LIN {X 0,Y 474.587,Z 604.783,A -85,B 0,C 180,E1 6633.911,E2 6633.911} C_VEL
LIN {X 0,Y 484.461,Z 641.921,A -85,B 0,C 180,E1 6635.452,E2 6635.452} C_VEL
LIN {X 0,Y 481.473,Z 693.679,A -85,B 0,C 180,E1 6638.347,E2 6638.347} C_VEL
LIN {X 0,Y 478.667,Z 736.366,A -85,B 0,C 180,E1 6642.712,E2 6642.712} C_VEL
LIN {X 0,Y 476.602,Z 767.326,A -85,B 0,C 180,E1 6648.057,E2 6648.057} C_VEL
LIN {X 0,Y 475.424,Z 786.828,A -85,B 0,C 180,E1 6654.507,E2 6654.507} C_VEL
LIN {X 0,Y 475.028,Z 791.676,A -85,B 0,C 180,E1 6660.917,E2 6660.917} C_VEL
LIN {X 0,Y 475.519,Z 782.888,A -85,B 0,C 180,E1 6667.335,E2 6667.335} C_VEL
LIN {X 0,Y 477.046,Z 759.466,A -85,B 0,C 180,E1 6673.569,E2 6673.569} C_VEL
LIN {X 0,Y 479.555,Z 723.123,A -85,B 0,C 180,E1 6678.814,E2 6678.814} C_VEL
LIN {X 0,Y 482.628,Z 675.847,A -85,B 0,C 180,E1 6682.718,E2 6682.718} C_VEL
LIN {X 0,Y 482.433,Z 629.842,A -85,B 0,C 180,E1 6684.849,E2 6684.849} C_VEL
LIN {X 0,Y 474.42,Z 602.81,A -85,B 0,C 180,E1 6686.158,E2 6686.158} C_VEL
LIN {X 0,Y 474.205,Z 602.81,A -85,B 0,C 180,E1 6696.301,E2 6696.301} C_VEL
LIN {X 0,Y 474.043,Z 602.81,A -85,B 0,C 180,E1 6706.534,E2 6706.534} C_VEL
LIN {X 0,Y 473.963,Z 602.81,A -85,B 0,C 180,E1 6707.161,E2 6707.161} C_VEL
LIN {X 0,Y 465.924,Z 602.81,A -85,B 0,C 180,E1 6711.395,E2 6711.395} C_VEL
LIN {X 0,Y 466.396,Z 602.81,A -85,B 0,C 180,E1 6721.87,E2 6721.87} C_VEL
LIN {X 0,Y 466.767,Z 604.8,A -85,B 0,C 180,E1 6722.959,E2 6722.959} C_VEL
LIN {X 0,Y 476.808,Z 643.163,A -85,B 0,C 180,E1 6724.21,E2 6724.21} C_VEL
LIN {X 0,Y 475.259,Z 703.396,A -85,B 0,C 180,E1 6725.752,E2 6725.752} C_VEL
LIN {X 0,Y 472.339,Z 755.137,A -85,B 0,C 180,E1 6729.032,E2 6729.032} C_VEL
LIN {X 0,Y 469.648,Z 797.381,A -85,B 0,C 180,E1 6733.842,E2 6733.842} C_VEL
LIN {X 0,Y 468.095,Z 827.68,A -85,B 0,C 180,E1 6739.745,E2 6739.745} C_VEL
LIN {X 0,Y 467.651,Z 842.415,A -85,B 0,C 180,E1 6745.362,E2 6745.362} C_VEL
LIN {X 0,Y 467.519,Z 845.96,A -85,B 0,C 180,E1 6750.945,E2 6750.945} C_VEL
LIN {X 0,Y 467.394,Z 838.979,A -85,B 0,C 180,E1 6756.54,E2 6756.54} C_VEL
LIN {X 0,Y 468.068,Z 818.515,A -85,B 0,C 180,E1 6762.593,E2 6762.593} C_VEL
LIN {X 0,Y 470.107,Z 786.148,A -85,B 0,C 180,E1 6767.872,E2 6767.872} C_VEL
LIN {X 0,Y 473.479,Z 740.316,A -85,B 0,C 180,E1 6772.26,E2 6772.26} C_VEL
LIN {X 0,Y 476.388,Z 687.666,A -85,B 0,C 180,E1 6774.942,E2 6774.942} C_VEL
LIN {X 0,Y 475.283,Z 629.797,A -85,B 0,C 180,E1 6776.245,E2 6776.245} C_VEL
LIN {X 0,Y 466.568,Z 602.81,A -85,B 0,C 180,E1 6777.358,E2 6777.358} C_VEL
LIN {X 0,Y 466.192,Z 602.81,A -85,B 0,C 180,E1 6787.107,E2 6787.107} C_VEL
LIN {X 0,Y 466.037,Z 602.81,A -85,B 0,C 180,E1 6797.125,E2 6797.125} C_VEL
LIN {X 0,Y 466.048,Z 602.81,A -85,B 0,C 180,E1 6807.502,E2 6807.502} C_VEL
LIN {X 0,Y 466.362,Z 602.81,A -85,B 0,C 180,E1 6818.055,E2 6818.055} C_VEL
LIN {X 0,Y 466.622,Z 604.64,A -85,B 0,C 180,E1 6823.647,E2 6823.647} C_VEL
LIN {X 0,Y 472.282,Z 636.649,A -85,B 0,C 180,E1 6825.408,E2 6825.408} C_VEL
LIN {X 0,Y 470.46,Z 672.434,A -85,B 0,C 180,E1 6828.604,E2 6828.604} C_VEL
LIN {X 0,Y 468.864,Z 697.709,A -85,B 0,C 180,E1 6833.027,E2 6833.027} C_VEL
LIN {X 0,Y 468.205,Z 708.246,A -85,B 0,C 180,E1 6837.212,E2 6837.212} C_VEL
LIN {X 0,Y 468.292,Z 707.263,A -85,B 0,C 180,E1 6842.785,E2 6842.785} C_VEL
LIN {X 0,Y 469.071,Z 690.988,A -85,B 0,C 180,E1 6847.901,E2 6847.901} C_VEL
LIN {X 0,Y 470.442,Z 661.657,A -85,B 0,C 180,E1 6852.101,E2 6852.101} C_VEL
LIN {X 0,Y 471.362,Z 621.95,A -85,B 0,C 180,E1 6854.97,E2 6854.97} C_VEL
LIN {X 0,Y 467.004,Z 602.81,A -85,B 0,C 180,E1 6856.032,E2 6856.032} C_VEL
LIN {X 0,Y 466.282,Z 602.81,A -85,B 0,C 180,E1 6866.471,E2 6866.471} C_VEL
LIN {X 0,Y 465.936,Z 602.81,A -85,B 0,C 180,E1 6877.048,E2 6877.048} C_VEL
LIN {X 0,Y 466.013,Z 602.81,A -85,B 0,C 180,E1 6887.108,E2 6887.108} C_VEL
LIN {X 0,Y 466.059,Z 602.81,A -85,B 0,C 180,E1 6897.489,E2 6897.489} C_VEL
LIN {X 0,Y 466.09,Z 602.81,A -85,B 0,C 180,E1 6905.971,E2 6905.971} C_VEL
LIN {X 0,Y 466.45,Z 602.81,A -85,B 0,C 180,E1 6915.863,E2 6915.863} C_VEL
LIN {X 0,Y 466.809,Z 602.81,A -85,B 0,C 180,E1 6925.324,E2 6925.324} C_VEL
LIN {X 0,Y 466.837,Z 602.81,A -85,B 0,C 180,E1 6932.779,E2 6932.779} C_VEL
LIN {X 0,Y 466.774,Z 602.81,A -85,B 0,C 180,E1 6942.183,E2 6942.183} C_VEL
LIN {X 0,Y 466.507,Z 602.81,A -85,B 0,C 180,E1 6952.023,E2 6952.023} C_VEL
LIN {X 0,Y 466.124,Z 602.81,A -85,B 0,C 180,E1 6962.47,E2 6962.47} C_VEL
LIN {X 0,Y 466.088,Z 602.81,A -85,B 0,C 180,E1 6972.902,E2 6972.902} C_VEL
LIN {X 0,Y 466.061,Z 602.81,A -85,B 0,C 180,E1 6982.963,E2 6982.963} C_VEL
LIN {X 0,Y 466.598,Z 604.805,A -85,B 0,C 180,E1 6993.49,E2 6993.49} C_VEL
LIN {X 0,Y 477.008,Z 643.776,A -85,B 0,C 180,E1 6995.156,E2 6995.156} C_VEL
LIN {X 0,Y 473.764,Z 696.064,A -85,B 0,C 180,E1 6998.193,E2 6998.193} C_VEL
LIN {X 0,Y 470.799,Z 738.175,A -85,B 0,C 180,E1 7002.655,E2 7002.655} C_VEL
LIN {X 0,Y 468.494,Z 769.542,A -85,B 0,C 180,E1 7008.322,E2 7008.322} C_VEL
LIN {X 0,Y 467.463,Z 787.235,A -85,B 0,C 180,E1 7014.413,E2 7014.413} C_VEL
LIN {X 0,Y 467.043,Z 792.143,A -85,B 0,C 180,E1 7020.932,E2 7020.932} C_VEL
LIN {X 0,Y 467.586,Z 783.317,A -85,B 0,C 180,E1 7027.46,E2 7027.46} C_VEL
LIN {X 0,Y 469.241,Z 759.761,A -85,B 0,C 180,E1 7033.8,E2 7033.8} C_VEL
LIN {X 0,Y 471.891,Z 723.653,A -85,B 0,C 180,E1 7039.082,E2 7039.082} C_VEL
LIN {X 0,Y 475.132,Z 676.627,A -85,B 0,C 180,E1 7043.033,E2 7043.033} C_VEL
LIN {X 0,Y 475.01,Z 631.363,A -85,B 0,C 180,E1 7045.198,E2 7045.198} C_VEL
LIN {X 0,Y 466.413,Z 602.81,A -85,B 0,C 180,E1 7046.571,E2 7046.571} C_VEL
LIN {X 0,Y 466.14,Z 602.81,A -85,B 0,C 180,E1 7057.132,E2 7057.132} C_VEL
LIN {X 0,Y 465.968,Z 602.81,A -85,B 0,C 180,E1 7067.153,E2 7067.153} C_VEL
LIN {X 0,Y 465.924,Z 602.81,A -85,B 0,C 180,E1 7071.395,E2 7071.395} C_VEL
LIN {X 0,Y 457.883,Z 602.81,A -85,B 0,C 180,E1 7075.697,E2 7075.697} C_VEL
LIN {X 0,Y 458.591,Z 604.397,A -85,B 0,C 180,E1 7082.413,E2 7082.413} C_VEL
LIN {X 0,Y 469.3,Z 643.439,A -85,B 0,C 180,E1 7083.879,E2 7083.879} C_VEL
LIN {X 0,Y 467.636,Z 703.35,A -85,B 0,C 180,E1 7085.454,E2 7085.454} C_VEL
LIN {X 0,Y 464.495,Z 754.843,A -85,B 0,C 180,E1 7088.795,E2 7088.795} C_VEL
LIN {X 0,Y 461.667,Z 797.815,A -85,B 0,C 180,E1 7093.793,E2 7093.793} C_VEL
LIN {X 0,Y 460.148,Z 827.011,A -85,B 0,C 180,E1 7099.566,E2 7099.566} C_VEL
LIN {X 0,Y 459.688,Z 841.908,A -85,B 0,C 180,E1 7105.282,E2 7105.282} C_VEL
LIN {X 0,Y 459.558,Z 845.507,A -85,B 0,C 180,E1 7110.961,E2 7110.961} C_VEL
LIN {X 0,Y 459.405,Z 836.974,A -85,B 0,C 180,E1 7117.313,E2 7117.313} C_VEL
LIN {X 0,Y 460.425,Z 814.602,A -85,B 0,C 180,E1 7123.519,E2 7123.519} C_VEL
LIN {X 0,Y 462.869,Z 778.456,A -85,B 0,C 180,E1 7129.028,E2 7129.028} C_VEL
LIN {X 0,Y 466.4,Z 732.254,A -85,B 0,C 180,E1 7133.123,E2 7133.123} C_VEL
LIN {X 0,Y 469.408,Z 678.55,A -85,B 0,C 180,E1 7135.577,E2 7135.577} C_VEL
LIN {X 0,Y 467.786,Z 630.643,A -85,B 0,C 180,E1 7136.631,E2 7136.631} C_VEL
LIN {X 0,Y 458.524,Z 602.81,A -85,B 0,C 180,E1 7137.747,E2 7137.747} C_VEL
LIN {X 0,Y 458.105,Z 602.81,A -85,B 0,C 180,E1 7148.88,E2 7148.88} C_VEL
LIN {X 0,Y 458.01,Z 602.81,A -85,B 0,C 180,E1 7158.218,E2 7158.218} C_VEL
LIN {X 0,Y 458.068,Z 602.81,A -85,B 0,C 180,E1 7169.102,E2 7169.102} C_VEL
LIN {X 0,Y 458.391,Z 602.81,A -85,B 0,C 180,E1 7179.658,E2 7179.658} C_VEL
LIN {X 0,Y 458.565,Z 604.492,A -85,B 0,C 180,E1 7183.224,E2 7183.224} C_VEL
LIN {X 0,Y 464.67,Z 638.988,A -85,B 0,C 180,E1 7185.202,E2 7185.202} C_VEL
LIN {X 0,Y 462.733,Z 675.713,A -85,B 0,C 180,E1 7188.651,E2 7188.651} C_VEL
LIN {X 0,Y 461.053,Z 699.023,A -85,B 0,C 180,E1 7192.909,E2 7192.909} C_VEL
LIN {X 0,Y 460.334,Z 709.509,A -85,B 0,C 180,E1 7197.164,E2 7197.164} C_VEL
LIN {X 0,Y 460.399,Z 708.377,A -85,B 0,C 180,E1 7202.832,E2 7202.832} C_VEL
LIN {X 0,Y 461.229,Z 691.913,A -85,B 0,C 180,E1 7208.036,E2 7208.036} C_VEL
LIN {X 0,Y 462.65,Z 662.358,A -85,B 0,C 180,E1 7212.308,E2 7212.308} C_VEL
LIN {X 0,Y 463.26,Z 621.442,A -85,B 0,C 180,E1 7215.288,E2 7215.288} C_VEL
LIN {X 0,Y 458.967,Z 602.81,A -85,B 0,C 180,E1 7216.32,E2 7216.32} C_VEL
LIN {X 0,Y 458.298,Z 602.81,A -85,B 0,C 180,E1 7226.55,E2 7226.55} C_VEL
LIN {X 0,Y 457.859,Z 602.81,A -85,B 0,C 180,E1 7235.688,E2 7235.688} C_VEL
LIN {X 0,Y 457.999,Z 602.81,A -85,B 0,C 180,E1 7245.425,E2 7245.425} C_VEL
LIN {X 0,Y 457.909,Z 602.81,A -85,B 0,C 180,E1 7254.538,E2 7254.538} C_VEL
LIN {X 0,Y 458.158,Z 602.81,A -85,B 0,C 180,E1 7263.425,E2 7263.425} C_VEL
LIN {X 0,Y 458.484,Z 602.81,A -85,B 0,C 180,E1 7273.646,E2 7273.646} C_VEL
LIN {X 0,Y 458.919,Z 602.81,A -85,B 0,C 180,E1 7283.339,E2 7283.339} C_VEL
LIN {X 0,Y 458.987,Z 602.81,A -85,B 0,C 180,E1 7290.932,E2 7290.932} C_VEL
LIN {X 0,Y 458.656,Z 602.81,A -85,B 0,C 180,E1 7300.468,E2 7300.468} C_VEL
LIN {X 0,Y 458.524,Z 602.81,A -85,B 0,C 180,E1 7310.316,E2 7310.316} C_VEL
LIN {X 0,Y 458.155,Z 602.81,A -85,B 0,C 180,E1 7320.869,E2 7320.869} C_VEL
LIN {X 0,Y 458.112,Z 602.81,A -85,B 0,C 180,E1 7330.211,E2 7330.211} C_VEL
LIN {X 0,Y 458.029,Z 602.81,A -85,B 0,C 180,E1 7339.758,E2 7339.758} C_VEL
LIN {X 0,Y 458.044,Z 602.81,A -85,B 0,C 180,E1 7349.104,E2 7349.104} C_VEL
LIN {X 0,Y 458.508,Z 604.691,A -85,B 0,C 180,E1 7353.053,E2 7353.053} C_VEL
LIN {X 0,Y 469.493,Z 645.825,A -85,B 0,C 180,E1 7354.861,E2 7354.861} C_VEL
LIN {X 0,Y 466.031,Z 698.135,A -85,B 0,C 180,E1 7358.011,E2 7358.011} C_VEL
LIN {X 0,Y 462.721,Z 741.624,A -85,B 0,C 180,E1 7362.835,E2 7362.835} C_VEL
LIN {X 0,Y 460.351,Z 771.752,A -85,B 0,C 180,E1 7368.594,E2 7368.594} C_VEL
LIN {X 0,Y 459.507,Z 787.639,A -85,B 0,C 180,E1 7374.316,E2 7374.316} C_VEL
LIN {X 0,Y 459.059,Z 792.609,A -85,B 0,C 180,E1 7380.949,E2 7380.949} C_VEL
LIN {X 0,Y 459.65,Z 783.832,A -85,B 0,C 180,E1 7387.557,E2 7387.557} C_VEL
LIN {X 0,Y 461.352,Z 760.714,A -85,B 0,C 180,E1 7393.915,E2 7393.915} C_VEL
LIN {X 0,Y 464.199,Z 724.52,A -85,B 0,C 180,E1 7399.33,E2 7399.33} C_VEL
LIN {X 0,Y 467.603,Z 678.481,A -85,B 0,C 180,E1 7403.299,E2 7403.299} C_VEL
LIN {X 0,Y 467.814,Z 633.482,A -85,B 0,C 180,E1 7405.532,E2 7405.532} C_VEL
LIN {X 0,Y 458.36,Z 602.81,A -85,B 0,C 180,E1 7407.078,E2 7407.078} C_VEL
LIN {X 0,Y 458.069,Z 602.81,A -85,B 0,C 180,E1 7417.799,E2 7417.799} C_VEL
LIN {X 0,Y 457.963,Z 602.81,A -85,B 0,C 180,E1 7428.208,E2 7428.208} C_VEL
LIN {X 0,Y 457.883,Z 602.81,A -85,B 0,C 180,E1 7435.697,E2 7435.697} C_VEL
LIN {X 0,Y 450.118,Z 602.81,A -85,B 0,C 180,E1 7440.088,E2 7440.088} C_VEL
LIN {X 0,Y 450.613,Z 604.727,A -85,B 0,C 180,E1 7441.849,E2 7441.849} C_VEL
LIN {X 0,Y 462.079,Z 643.809,A -85,B 0,C 180,E1 7443.466,E2 7443.466} C_VEL
LIN {X 0,Y 459.911,Z 705.455,A -85,B 0,C 180,E1 7445.259,E2 7445.259} C_VEL
LIN {X 0,Y 456.642,Z 755.376,A -85,B 0,C 180,E1 7448.632,E2 7448.632} C_VEL
LIN {X 0,Y 453.79,Z 796.99,A -85,B 0,C 180,E1 7453.504,E2 7453.504} C_VEL
LIN {X 0,Y 452.226,Z 826.375,A -85,B 0,C 180,E1 7459.382,E2 7459.382} C_VEL
LIN {X 0,Y 451.706,Z 841.4,A -85,B 0,C 180,E1 7465.198,E2 7465.198} C_VEL
LIN {X 0,Y 451.566,Z 845.053,A -85,B 0,C 180,E1 7470.978,E2 7470.978} C_VEL
LIN {X 0,Y 451.422,Z 836.605,A -85,B 0,C 180,E1 7477.395,E2 7477.395} C_VEL
LIN {X 0,Y 452.517,Z 813.985,A -85,B 0,C 180,E1 7483.76,E2 7483.76} C_VEL
LIN {X 0,Y 455.152,Z 777.615,A -85,B 0,C 180,E1 7489.364,E2 7489.364} C_VEL
LIN {X 0,Y 458.866,Z 730.967,A -85,B 0,C 180,E1 7493.525,E2 7493.525} C_VEL
LIN {X 0,Y 462.008,Z 677.666,A -85,B 0,C 180,E1 7495.97,E2 7495.97} C_VEL
LIN {X 0,Y 460.582,Z 632.598,A -85,B 0,C 180,E1 7496.986,E2 7496.986} C_VEL
LIN {X 0,Y 450.482,Z 602.81,A -85,B 0,C 180,E1 7498.134,E2 7498.134} C_VEL
LIN {X 0,Y 450.094,Z 602.81,A -85,B 0,C 180,E1 7508.605,E2 7508.605} C_VEL
LIN {X 0,Y 450.008,Z 602.81,A -85,B 0,C 180,E1 7519.371,E2 7519.371} C_VEL
LIN {X 0,Y 450.045,Z 602.81,A -85,B 0,C 180,E1 7529.319,E2 7529.319} C_VEL
LIN {X 0,Y 450.325,Z 602.81,A -85,B 0,C 180,E1 7539.277,E2 7539.277} C_VEL
LIN {X 0,Y 450.601,Z 604.68,A -85,B 0,C 180,E1 7542.785,E2 7542.785} C_VEL
LIN {X 0,Y 457.176,Z 639.418,A -85,B 0,C 180,E1 7544.848,E2 7544.848} C_VEL
LIN {X 0,Y 455.065,Z 675.382,A -85,B 0,C 180,E1 7548.213,E2 7548.213} C_VEL
LIN {X 0,Y 453.228,Z 700.391,A -85,B 0,C 180,E1 7552.786,E2 7552.786} C_VEL
LIN {X 0,Y 452.449,Z 710.775,A -85,B 0,C 180,E1 7557.115,E2 7557.115} C_VEL
LIN {X 0,Y 452.487,Z 709.488,A -85,B 0,C 180,E1 7562.882,E2 7562.882} C_VEL
LIN {X 0,Y 453.377,Z 692.765,A -85,B 0,C 180,E1 7568.177,E2 7568.177} C_VEL
LIN {X 0,Y 454.86,Z 662.916,A -85,B 0,C 180,E1 7572.522,E2 7572.522} C_VEL
LIN {X 0,Y 455.335,Z 621.95,A -85,B 0,C 180,E1 7575.545,E2 7575.545} C_VEL
LIN {X 0,Y 450.908,Z 602.81,A -85,B 0,C 180,E1 7576.62,E2 7576.62} C_VEL
LIN {X 0,Y 450.218,Z 602.81,A -85,B 0,C 180,E1 7587.065,E2 7587.065} C_VEL
LIN {X 0,Y 449.824,Z 602.81,A -85,B 0,C 180,E1 7597.535,E2 7597.535} C_VEL
LIN {X 0,Y 449.953,Z 602.81,A -85,B 0,C 180,E1 7606.474,E2 7606.474} C_VEL
LIN {X 0,Y 449.922,Z 602.81,A -85,B 0,C 180,E1 7616.17,E2 7616.17} C_VEL
LIN {X 0,Y 450.038,Z 602.81,A -85,B 0,C 180,E1 7625.056,E2 7625.056} C_VEL
LIN {X 0,Y 450.406,Z 602.81,A -85,B 0,C 180,E1 7635.348,E2 7635.348} C_VEL
LIN {X 0,Y 450.799,Z 602.81,A -85,B 0,C 180,E1 7645.157,E2 7645.157} C_VEL
LIN {X 0,Y 450.85,Z 602.81,A -85,B 0,C 180,E1 7652.878,E2 7652.878} C_VEL
LIN {X 0,Y 450.75,Z 602.81,A -85,B 0,C 180,E1 7662.623,E2 7662.623} C_VEL
LIN {X 0,Y 450.399,Z 602.81,A -85,B 0,C 180,E1 7672.777,E2 7672.777} C_VEL
LIN {X 0,Y 450.136,Z 602.81,A -85,B 0,C 180,E1 7681.481,E2 7681.481} C_VEL
LIN {X 0,Y 450.068,Z 602.81,A -85,B 0,C 180,E1 7691.083,E2 7691.083} C_VEL
LIN {X 0,Y 449.986,Z 602.81,A -85,B 0,C 180,E1 7701.403,E2 7701.403} C_VEL
LIN {X 0,Y 450.311,Z 603.715,A -85,B 0,C 180,E1 7712.581,E2 7712.581} C_VEL
LIN {X 0,Y 462.046,Z 647.117,A -85,B 0,C 180,E1 7714.533,E2 7714.533} C_VEL
LIN {X 0,Y 458.435,Z 698.698,A -85,B 0,C 180,E1 7717.711,E2 7717.711} C_VEL
LIN {X 0,Y 454.996,Z 741.752,A -85,B 0,C 180,E1 7722.547,E2 7722.547} C_VEL
LIN {X 0,Y 452.5,Z 772.015,A -85,B 0,C 180,E1 7728.394,E2 7728.394} C_VEL
LIN {X 0,Y 451.347,Z 789.632,A -85,B 0,C 180,E1 7735.18,E2 7735.18} C_VEL
LIN {X 0,Y 451.075,Z 793.077,A -85,B 0,C 180,E1 7740.965,E2 7740.965} C_VEL
LIN {X 0,Y 451.686,Z 784.691,A -85,B 0,C 180,E1 7747.516,E2 7747.516} C_VEL
LIN {X 0,Y 453.316,Z 763.034,A -85,B 0,C 180,E1 7753.766,E2 7753.766} C_VEL
LIN {X 0,Y 456.314,Z 727.92,A -85,B 0,C 180,E1 7759.299,E2 7759.299} C_VEL
LIN {X 0,Y 459.952,Z 682.313,A -85,B 0,C 180,E1 7763.453,E2 7763.453} C_VEL
LIN {X 0,Y 460.331,Z 634.38,A -85,B 0,C 180,E1 7765.95,E2 7765.95} C_VEL
LIN {X 0,Y 450.345,Z 602.81,A -85,B 0,C 180,E1 7767.655,E2 7767.655} C_VEL
LIN {X 0,Y 450.046,Z 602.81,A -85,B 0,C 180,E1 7778.595,E2 7778.595} C_VEL
LIN {X 0,Y 449.946,Z 602.81,A -85,B 0,C 180,E1 7789.363,E2 7789.363} C_VEL
LIN {X 0,Y 450.118,Z 602.81,A -85,B 0,C 180,E1 7800.088,E2 7800.088} C_VEL
LIN {X 0,Y 450.058,Z 611.324,A -85,B 0,C 180,E1 7801.586,E2 7801.586} C_VEL
LIN {X 0,Y 452.222,Z 631.755,A -85,B 0,C 180,E1 7802.579,E2 7802.579} C_VEL
LIN {X 0,Y 454.672,Z 660.701,A -85,B 0,C 180,E1 7803.365,E2 7803.365} C_VEL
LIN {X 0,Y 451.664,Z 717.922,A -85,B 0,C 180,E1 7805.584,E2 7805.584} C_VEL
LIN {X 0,Y 447.917,Z 767.78,A -85,B 0,C 180,E1 7809.57,E2 7809.57} C_VEL
LIN {X 0,Y 445.044,Z 806.637,A -85,B 0,C 180,E1 7814.948,E2 7814.948} C_VEL
LIN {X 0,Y 443.683,Z 832.146,A -85,B 0,C 180,E1 7821.163,E2 7821.163} C_VEL
LIN {X 0,Y 443.497,Z 843.283,A -85,B 0,C 180,E1 7827.074,E2 7827.074} C_VEL
LIN {X 0,Y 443.803,Z 842.439,A -85,B 0,C 180,E1 7833.937,E2 7833.937} C_VEL
LIN {X 0,Y 444.078,Z 826.443,A -85,B 0,C 180,E1 7840.848,E2 7840.848} C_VEL
LIN {X 0,Y 445.958,Z 795.95,A -85,B 0,C 180,E1 7847.102,E2 7847.102} C_VEL
LIN {X 0,Y 449.574,Z 753.959,A -85,B 0,C 180,E1 7852.049,E2 7852.049} C_VEL
LIN {X 0,Y 453.219,Z 702.319,A -85,B 0,C 180,E1 7855.444,E2 7855.444} C_VEL
LIN {X 0,Y 454.369,Z 638.475,A -85,B 0,C 180,E1 7857.215,E2 7857.215} C_VEL
LIN {X 0,Y 442.327,Z 602.81,A -85,B 0,C 180,E1 7858.811,E2 7858.811} C_VEL
LIN {X 0,Y 442.036,Z 602.81,A -85,B 0,C 180,E1 7869.444,E2 7869.444} C_VEL
LIN {X 0,Y 441.914,Z 602.81,A -85,B 0,C 180,E1 7877.961,E2 7877.961} C_VEL
LIN {X 0,Y 441.919,Z 602.81,A -85,B 0,C 180,E1 7887.841,E2 7887.841} C_VEL
LIN {X 0,Y 442.292,Z 602.81,A -85,B 0,C 180,E1 7898.883,E2 7898.883} C_VEL
LIN {X 0,Y 442.515,Z 604.411,A -85,B 0,C 180,E1 7902.298,E2 7902.298} C_VEL
LIN {X 0,Y 449.707,Z 640.311,A -85,B 0,C 180,E1 7904.51,E2 7904.51} C_VEL
LIN {X 0,Y 447.416,Z 676.976,A -85,B 0,C 180,E1 7908.009,E2 7908.009} C_VEL
LIN {X 0,Y 445.412,Z 701.788,A -85,B 0,C 180,E1 7912.658,E2 7912.658} C_VEL
LIN {X 0,Y 444.591,Z 712.065,A -85,B 0,C 180,E1 7917.064,E2 7917.064} C_VEL
LIN {X 0,Y 444.575,Z 710.597,A -85,B 0,C 180,E1 7922.933,E2 7922.933} C_VEL
LIN {X 0,Y 445.507,Z 693.633,A -85,B 0,C 180,E1 7928.322,E2 7928.322} C_VEL
LIN {X 0,Y 447.08,Z 663.468,A -85,B 0,C 180,E1 7932.744,E2 7932.744} C_VEL
LIN {X 0,Y 447.561,Z 623.187,A -85,B 0,C 180,E1 7935.769,E2 7935.769} C_VEL
LIN {X 0,Y 442.822,Z 602.81,A -85,B 0,C 180,E1 7936.933,E2 7936.933} C_VEL
LIN {X 0,Y 442.131,Z 602.81,A -85,B 0,C 180,E1 7947.601,E2 7947.601} C_VEL
LIN {X 0,Y 441.795,Z 602.81,A -85,B 0,C 180,E1 7956.946,E2 7956.946} C_VEL
LIN {X 0,Y 441.85,Z 602.81,A -85,B 0,C 180,E1 7967.592,E2 7967.592} C_VEL
LIN {X 0,Y 441.9,Z 602.81,A -85,B 0,C 180,E1 7977.825,E2 7977.825} C_VEL
LIN {X 0,Y 441.906,Z 602.81,A -85,B 0,C 180,E1 7986.725,E2 7986.725} C_VEL
LIN {X 0,Y 442.419,Z 602.81,A -85,B 0,C 180,E1 7997.102,E2 7997.102} C_VEL
LIN {X 0,Y 443.065,Z 602.81,A -85,B 0,C 180,E1 8007.039,E2 8007.039} C_VEL
LIN {X 0,Y 443.053,Z 602.81,A -85,B 0,C 180,E1 8016.868,E2 8016.868} C_VEL
LIN {X 0,Y 442.453,Z 602.81,A -85,B 0,C 180,E1 8026.931,E2 8026.931} C_VEL
LIN {X 0,Y 442.197,Z 602.81,A -85,B 0,C 180,E1 8037.578,E2 8037.578} C_VEL
LIN {X 0,Y 442.065,Z 602.81,A -85,B 0,C 180,E1 8046.898,E2 8046.898} C_VEL
LIN {X 0,Y 441.888,Z 602.81,A -85,B 0,C 180,E1 8057.56,E2 8057.56} C_VEL
LIN {X 0,Y 441.91,Z 602.81,A -85,B 0,C 180,E1 8067.844,E2 8067.844} C_VEL
LIN {X 0,Y 442.355,Z 604.215,A -85,B 0,C 180,E1 8072.144,E2 8072.144} C_VEL
LIN {X 0,Y 454.587,Z 648.388,A -85,B 0,C 180,E1 8074.205,E2 8074.205} C_VEL
LIN {X 0,Y 450.707,Z 700.968,A -85,B 0,C 180,E1 8077.56,E2 8077.56} C_VEL
LIN {X 0,Y 447.031,Z 743.825,A -85,B 0,C 180,E1 8082.554,E2 8082.554} C_VEL
LIN {X 0,Y 444.383,Z 774.044,A -85,B 0,C 180,E1 8088.678,E2 8088.678} C_VEL
LIN {X 0,Y 443.405,Z 790.036,A -85,B 0,C 180,E1 8095.093,E2 8095.093} C_VEL
LIN {X 0,Y 443.091,Z 793.55,A -85,B 0,C 180,E1 8100.983,E2 8100.983} C_VEL
LIN {X 0,Y 443.699,Z 785.6,A -85,B 0,C 180,E1 8107.463,E2 8107.463} C_VEL
LIN {X 0,Y 445.508,Z 763.647,A -85,B 0,C 180,E1 8113.974,E2 8113.974} C_VEL
LIN {X 0,Y 448.74,Z 728.276,A -85,B 0,C 180,E1 8119.638,E2 8119.638} C_VEL
LIN {X 0,Y 452.625,Z 682.616,A -85,B 0,C 180,E1 8123.856,E2 8123.856} C_VEL
LIN {X 0,Y 453.175,Z 636.433,A -85,B 0,C 180,E1 8126.334,E2 8126.334} C_VEL
LIN {X 0,Y 442.283,Z 602.81,A -85,B 0,C 180,E1 8128.176,E2 8128.176} C_VEL
LIN {X 0,Y 441.991,Z 602.81,A -85,B 0,C 180,E1 8139.453,E2 8139.453} C_VEL
LIN {X 0,Y 441.839,Z 602.81,A -85,B 0,C 180,E1 8147.98,E2 8147.98} C_VEL
LIN {X 0,Y 441.941,Z 602.81,A -85,B 0,C 180,E1 8157.866,E2 8157.866} C_VEL
LIN {X 0,Y 442.419,Z 604.32,A -85,B 0,C 180,E1 8161.202,E2 8161.202} C_VEL
LIN {X 0,Y 452.222,Z 631.755,A -85,B 0,C 180,E1 8162.579,E2 8162.579} C_VEL
LIN {X 0,Y 448.775,Z 658.085,A -85,B 0,C 180,E1 8162.914,E2 8162.914} C_VEL
LIN {X 0,Y 447.31,Z 667.064,A -85,B 0,C 180,E1 8163.062,E2 8163.062} C_VEL
LIN {X 0,Y 443.81,Z 723.189,A -85,B 0,C 180,E1 8165.527,E2 8165.527} C_VEL
LIN {X 0,Y 439.685,Z 772.638,A -85,B 0,C 180,E1 8169.829,E2 8169.829} C_VEL
LIN {X 0,Y 436.768,Z 809.92,A -85,B 0,C 180,E1 8175.429,E2 8175.429} C_VEL
LIN {X 0,Y 435.643,Z 833.026,A -85,B 0,C 180,E1 8181.504,E2 8181.504} C_VEL
LIN {X 0,Y 435.51,Z 842.811,A -85,B 0,C 180,E1 8187.021,E2 8187.021} C_VEL
LIN {X 0,Y 435.809,Z 841.965,A -85,B 0,C 180,E1 8194.009,E2 8194.009} C_VEL
LIN {X 0,Y 436.067,Z 825.849,A -85,B 0,C 180,E1 8201.05,E2 8201.05} C_VEL
LIN {X 0,Y 438.066,Z 795.441,A -85,B 0,C 180,E1 8207.373,E2 8207.373} C_VEL
LIN {X 0,Y 441.95,Z 753.031,A -85,B 0,C 180,E1 8212.423,E2 8212.423} C_VEL
LIN {X 0,Y 445.789,Z 701.647,A -85,B 0,C 180,E1 8215.836,E2 8215.836} C_VEL
LIN {X 0,Y 446.615,Z 638.436,A -85,B 0,C 180,E1 8217.645,E2 8217.645} C_VEL
LIN {X 0,Y 434.261,Z 602.81,A -85,B 0,C 180,E1 8219.306,E2 8219.306} C_VEL
LIN {X 0,Y 433.915,Z 602.81,A -85,B 0,C 180,E1 8230.332,E2 8230.332} C_VEL
LIN {X 0,Y 433.833,Z 602.81,A -85,B 0,C 180,E1 8239.675,E2 8239.675} C_VEL
LIN {X 0,Y 433.941,Z 602.81,A -85,B 0,C 180,E1 8249.53,E2 8249.53} C_VEL
LIN {X 0,Y 434.27,Z 602.81,A -85,B 0,C 180,E1 8260.611,E2 8260.611} C_VEL
LIN {X 0,Y 434.533,Z 604.508,A -85,B 0,C 180,E1 8261.785,E2 8261.785} C_VEL
LIN {X 0,Y 442.314,Z 640.952,A -85,B 0,C 180,E1 8264.125,E2 8264.125} C_VEL
LIN {X 0,Y 439.764,Z 678.633,A -85,B 0,C 180,E1 8267.797,E2 8267.797} C_VEL
LIN {X 0,Y 437.601,Z 703.657,A -85,B 0,C 180,E1 8272.659,E2 8272.659} C_VEL
LIN {X 0,Y 436.732,Z 713.365,A -85,B 0,C 180,E1 8277.011,E2 8277.011} C_VEL
LIN {X 0,Y 436.663,Z 711.695,A -85,B 0,C 180,E1 8282.986,E2 8282.986} C_VEL
LIN {X 0,Y 437.582,Z 694.803,A -85,B 0,C 180,E1 8288.404,E2 8288.404} C_VEL
LIN {X 0,Y 439.202,Z 665.177,A -85,B 0,C 180,E1 8292.85,E2 8292.85} C_VEL
LIN {X 0,Y 439.878,Z 624.842,A -85,B 0,C 180,E1 8295.971,E2 8295.971} C_VEL
LIN {X 0,Y 434.741,Z 602.81,A -85,B 0,C 180,E1 8297.258,E2 8297.258} C_VEL
LIN {X 0,Y 434.09,Z 602.81,A -85,B 0,C 180,E1 8308.158,E2 8308.158} C_VEL
LIN {X 0,Y 433.731,Z 602.81,A -85,B 0,C 180,E1 8318.055,E2 8318.055} C_VEL
LIN {X 0,Y 433.769,Z 602.81,A -85,B 0,C 180,E1 8328.774,E2 8328.774} C_VEL
LIN {X 0,Y 433.899,Z 602.81,A -85,B 0,C 180,E1 8339.512,E2 8339.512} C_VEL
LIN {X 0,Y 434.08,Z 602.81,A -85,B 0,C 180,E1 8350.588,E2 8350.588} C_VEL
LIN {X 0,Y 434.851,Z 602.81,A -85,B 0,C 180,E1 8360.949,E2 8360.949} C_VEL
LIN {X 0,Y 434.997,Z 602.81,A -85,B 0,C 180,E1 8370.983,E2 8370.983} C_VEL
LIN {X 0,Y 434.644,Z 602.81,A -85,B 0,C 180,E1 8381.053,E2 8381.053} C_VEL
LIN {X 0,Y 434.371,Z 602.81,A -85,B 0,C 180,E1 8391.5,E2 8391.5} C_VEL
LIN {X 0,Y 433.996,Z 602.81,A -85,B 0,C 180,E1 8401.061,E2 8401.061} C_VEL
LIN {X 0,Y 433.907,Z 602.81,A -85,B 0,C 180,E1 8411.247,E2 8411.247} C_VEL
LIN {X 0,Y 433.858,Z 602.81,A -85,B 0,C 180,E1 8422.262,E2 8422.262} C_VEL
LIN {X 0,Y 434.218,Z 603.573,A -85,B 0,C 180,E1 8431.664,E2 8431.664} C_VEL
LIN {X 0,Y 447.04,Z 650.711,A -85,B 0,C 180,E1 8433.921,E2 8433.921} C_VEL
LIN {X 0,Y 443.099,Z 701.672,A -85,B 0,C 180,E1 8437.265,E2 8437.265} C_VEL
LIN {X 0,Y 439.213,Z 744.717,A -85,B 0,C 180,E1 8442.384,E2 8442.384} C_VEL
LIN {X 0,Y 436.522,Z 774.281,A -85,B 0,C 180,E1 8448.471,E2 8448.471} C_VEL
LIN {X 0,Y 435.432,Z 790.432,A -85,B 0,C 180,E1 8455.003,E2 8455.003} C_VEL
LIN {X 0,Y 435.107,Z 794.026,A -85,B 0,C 180,E1 8461.001,E2 8461.001} C_VEL
LIN {X 0,Y 435.869,Z 785.409,A -85,B 0,C 180,E1 8467.906,E2 8467.906} C_VEL
LIN {X 0,Y 437.926,Z 762.81,A -85,B 0,C 180,E1 8474.502,E2 8474.502} C_VEL
LIN {X 0,Y 441.377,Z 726.643,A -85,B 0,C 180,E1 8480.242,E2 8480.242} C_VEL
LIN {X 0,Y 445.607,Z 679.426,A -85,B 0,C 180,E1 8484.523,E2 8484.523} C_VEL
LIN {X 0,Y 445.952,Z 637.814,A -85,B 0,C 180,E1 8486.777,E2 8486.777} C_VEL
LIN {X 0,Y 434.185,Z 602.81,A -85,B 0,C 180,E1 8488.876,E2 8488.876} C_VEL
LIN {X 0,Y 433.928,Z 602.81,A -85,B 0,C 180,E1 8498.141,E2 8498.141} C_VEL
LIN {X 0,Y 433.783,Z 602.81,A -85,B 0,C 180,E1 8508.777,E2 8508.777} C_VEL
LIN {X 0,Y 434.008,Z 602.81,A -85,B 0,C 180,E1 8519.559,E2 8519.559} C_VEL
LIN {X 0,Y 434.464,Z 604.927,A -85,B 0,C 180,E1 8520.537,E2 8520.537} C_VEL
LIN {X 0,Y 447.68,Z 642.724,A -85,B 0,C 180,E1 8522.509,E2 8522.509} C_VEL
LIN {X 0,Y 447.31,Z 667.064,A -85,B 0,C 180,E1 8523.062,E2 8523.062} C_VEL
LIN {X 0,Y 438.142,Z 700.801,A -85,B 0,C 180,E1 8523.851,E2 8523.851} C_VEL
LIN {X 0,Y 433.834,Z 753.152,A -85,B 0,C 180,E1 8527.487,E2 8527.487} C_VEL
LIN {X 0,Y 430.127,Z 796.405,A -85,B 0,C 180,E1 8532.833,E2 8532.833} C_VEL
LIN {X 0,Y 428.222,Z 826.365,A -85,B 0,C 180,E1 8539.296,E2 8539.296} C_VEL
LIN {X 0,Y 427.642,Z 841.276,A -85,B 0,C 180,E1 8545.947,E2 8545.947} C_VEL
LIN {X 0,Y 427.62,Z 843.675,A -85,B 0,C 180,E1 8551.033,E2 8551.033} C_VEL
LIN {X 0,Y 427.483,Z 835.391,A -85,B 0,C 180,E1 8557.666,E2 8557.666} C_VEL
LIN {X 0,Y 428.799,Z 812.79,A -85,B 0,C 180,E1 8564.359,E2 8564.359} C_VEL
LIN {X 0,Y 432.02,Z 775.764,A -85,B 0,C 180,E1 8570.311,E2 8570.311} C_VEL
LIN {X 0,Y 436.27,Z 728.577,A -85,B 0,C 180,E1 8574.671,E2 8574.671} C_VEL
LIN {X 0,Y 439.961,Z 674.108,A -85,B 0,C 180,E1 8577.216,E2 8577.216} C_VEL
LIN {X 0,Y 438.377,Z 636.712,A -85,B 0,C 180,E1 8578.146,E2 8578.146} C_VEL
LIN {X 0,Y 426.195,Z 602.81,A -85,B 0,C 180,E1 8579.739,E2 8579.739} C_VEL
LIN {X 0,Y 425.933,Z 602.81,A -85,B 0,C 180,E1 8591.25,E2 8591.25} C_VEL
LIN {X 0,Y 425.804,Z 602.81,A -85,B 0,C 180,E1 8601.414,E2 8601.414} C_VEL
LIN {X 0,Y 425.925,Z 602.81,A -85,B 0,C 180,E1 8611.249,E2 8611.249} C_VEL
LIN {X 0,Y 426.456,Z 604.319,A -85,B 0,C 180,E1 8621.21,E2 8621.21} C_VEL
LIN {X 0,Y 434.883,Z 642.952,A -85,B 0,C 180,E1 8623.82,E2 8623.82} C_VEL
LIN {X 0,Y 432.151,Z 680.382,A -85,B 0,C 180,E1 8627.578,E2 8627.578} C_VEL
LIN {X 0,Y 429.826,Z 705.135,A -85,B 0,C 180,E1 8632.525,E2 8632.525} C_VEL
LIN {X 0,Y 428.855,Z 714.682,A -85,B 0,C 180,E1 8636.956,E2 8636.956} C_VEL
LIN {X 0,Y 428.772,Z 712.784,A -85,B 0,C 180,E1 8643.041,E2 8643.041} C_VEL
LIN {X 0,Y 429.702,Z 695.582,A -85,B 0,C 180,E1 8648.559,E2 8648.559} C_VEL
LIN {X 0,Y 431.418,Z 665.581,A -85,B 0,C 180,E1 8653.086,E2 8653.086} C_VEL
LIN {X 0,Y 431.752,Z 624.602,A -85,B 0,C 180,E1 8656.285,E2 8656.285} C_VEL
LIN {X 0,Y 426.662,Z 602.81,A -85,B 0,C 180,E1 8657.595,E2 8657.595} C_VEL
LIN {X 0,Y 425.996,Z 602.81,A -85,B 0,C 180,E1 8668.742,E2 8668.742} C_VEL
LIN {X 0,Y 425.732,Z 602.81,A -85,B 0,C 180,E1 8679.953,E2 8679.953} C_VEL
LIN {X 0,Y 425.699,Z 602.81,A -85,B 0,C 180,E1 8690.03,E2 8690.03} C_VEL
LIN {X 0,Y 425.895,Z 602.81,A -85,B 0,C 180,E1 8701.232,E2 8701.232} C_VEL
LIN {X 0,Y 426.21,Z 602.81,A -85,B 0,C 180,E1 8712.368,E2 8712.368} C_VEL
LIN {X 0,Y 426.899,Z 602.81,A -85,B 0,C 180,E1 8722.837,E2 8722.837} C_VEL
LIN {X 0,Y 427.006,Z 602.81,A -85,B 0,C 180,E1 8731.001,E2 8731.001} C_VEL
LIN {X 0,Y 426.623,Z 602.81,A -85,B 0,C 180,E1 8741.264,E2 8741.264} C_VEL
LIN {X 0,Y 426.329,Z 602.81,A -85,B 0,C 180,E1 8751.927,E2 8751.927} C_VEL
LIN {X 0,Y 425.961,Z 602.81,A -85,B 0,C 180,E1 8763.159,E2 8763.159} C_VEL
LIN {X 0,Y 425.879,Z 602.81,A -85,B 0,C 180,E1 8773.985,E2 8773.985} C_VEL
LIN {X 0,Y 425.789,Z 602.81,A -85,B 0,C 180,E1 8783.984,E2 8783.984} C_VEL
LIN {X 0,Y 426.343,Z 604.658,A -85,B 0,C 180,E1 8791.224,E2 8791.224} C_VEL
LIN {X 0,Y 439.6,Z 651.401,A -85,B 0,C 180,E1 8793.556,E2 8793.556} C_VEL
LIN {X 0,Y 435.376,Z 703.609,A -85,B 0,C 180,E1 8797.084,E2 8797.084} C_VEL
LIN {X 0,Y 431.326,Z 746.079,A -85,B 0,C 180,E1 8802.288,E2 8802.288} C_VEL
LIN {X 0,Y 428.392,Z 776.261,A -85,B 0,C 180,E1 8808.767,E2 8808.767} C_VEL
LIN {X 0,Y 427.47,Z 790.815,A -85,B 0,C 180,E1 8814.91,E2 8814.91} C_VEL
LIN {X 0,Y 427.131,Z 794.507,A -85,B 0,C 180,E1 8821.019,E2 8821.019} C_VEL
LIN {X 0,Y 427.975,Z 785.708,A -85,B 0,C 180,E1 8828.155,E2 8828.155} C_VEL
LIN {X 0,Y 430.248,Z 762.843,A -85,B 0,C 180,E1 8834.875,E2 8834.875} C_VEL
LIN {X 0,Y 433.859,Z 727.194,A -85,B 0,C 180,E1 8840.608,E2 8840.608} C_VEL
LIN {X 0,Y 438.363,Z 680.102,A -85,B 0,C 180,E1 8844.956,E2 8844.956} C_VEL
LIN {X 0,Y 438.751,Z 639.172,A -85,B 0,C 180,E1 8847.251,E2 8847.251} C_VEL
LIN {X 0,Y 426.101,Z 602.81,A -85,B 0,C 180,E1 8849.684,E2 8849.684} C_VEL
LIN {X 0,Y 425.872,Z 602.81,A -85,B 0,C 180,E1 8860.027,E2 8860.027} C_VEL
LIN {X 0,Y 425.755,Z 602.81,A -85,B 0,C 180,E1 8870.026,E2 8870.026} C_VEL
LIN {X 0,Y 426.189,Z 604.198,A -85,B 0,C 180,E1 8879.744,E2 8879.744} C_VEL
LIN {X 0,Y 440.495,Z 643.74,A -85,B 0,C 180,E1 8882.015,E2 8882.015} C_VEL
LIN {X 0,Y 438.142,Z 700.801,A -85,B 0,C 180,E1 8883.851,E2 8883.851} C_VEL
LIN {X 0,Y 428.152,Z 732.792,A -85,B 0,C 180,E1 8885.387,E2 8885.387} C_VEL
LIN {X 0,Y 423.465,Z 779.729,A -85,B 0,C 180,E1 8890.116,E2 8890.116} C_VEL
LIN {X 0,Y 420.534,Z 814.832,A -85,B 0,C 180,E1 8896.187,E2 8896.187} C_VEL
LIN {X 0,Y 419.695,Z 835.647,A -85,B 0,C 180,E1 8902.747,E2 8902.747} C_VEL
LIN {X 0,Y 419.875,Z 843.155,A -85,B 0,C 180,E1 8908.982,E2 8908.982} C_VEL
LIN {X 0,Y 419.582,Z 838.458,A -85,B 0,C 180,E1 8915.955,E2 8915.955} C_VEL
LIN {X 0,Y 420.164,Z 820.403,A -85,B 0,C 180,E1 8922.637,E2 8922.637} C_VEL
LIN {X 0,Y 422.853,Z 788.299,A -85,B 0,C 180,E1 8928.859,E2 8928.859} C_VEL
LIN {X 0,Y 427.283,Z 743.841,A -85,B 0,C 180,E1 8933.843,E2 8933.843} C_VEL
LIN {X 0,Y 431.609,Z 690.368,A -85,B 0,C 180,E1 8937.065,E2 8937.065} C_VEL
LIN {X 0,Y 431.314,Z 639.351,A -85,B 0,C 180,E1 8938.499,E2 8938.499} C_VEL
LIN {X 0,Y 418.167,Z 602.81,A -85,B 0,C 180,E1 8940.24,E2 8940.24} C_VEL
LIN {X 0,Y 417.871,Z 602.81,A -85,B 0,C 180,E1 8949.476,E2 8949.476} C_VEL
LIN {X 0,Y 417.786,Z 602.81,A -85,B 0,C 180,E1 8960.531,E2 8960.531} C_VEL
LIN {X 0,Y 417.904,Z 602.81,A -85,B 0,C 180,E1 8970.644,E2 8970.644} C_VEL
LIN {X 0,Y 418.42,Z 604.278,A -85,B 0,C 180,E1 8980.592,E2 8980.592} C_VEL
LIN {X 0,Y 427.67,Z 642.613,A -85,B 0,C 180,E1 8983.315,E2 8983.315} C_VEL
LIN {X 0,Y 424.706,Z 680.346,A -85,B 0,C 180,E1 8987.095,E2 8987.095} C_VEL
LIN {X 0,Y 422.109,Z 704.93,A -85,B 0,C 180,E1 8991.863,E2 8991.863} C_VEL
LIN {X 0,Y 420.998,Z 716.02,A -85,B 0,C 180,E1 8996.899,E2 8996.899} C_VEL
LIN {X 0,Y 420.858,Z 713.867,A -85,B 0,C 180,E1 9003.099,E2 9003.099} C_VEL
LIN {X 0,Y 421.846,Z 696.281,A -85,B 0,C 180,E1 9008.74,E2 9008.74} C_VEL
LIN {X 0,Y 423.702,Z 664.739,A -85,B 0,C 180,E1 9013.46,E2 9013.46} C_VEL
LIN {X 0,Y 423.875,Z 625.383,A -85,B 0,C 180,E1 9016.545,E2 9016.545} C_VEL
LIN {X 0,Y 418.595,Z 602.81,A -85,B 0,C 180,E1 9017.945,E2 9017.945} C_VEL
LIN {X 0,Y 417.96,Z 602.81,A -85,B 0,C 180,E1 9029.348,E2 9029.348} C_VEL
LIN {X 0,Y 417.705,Z 602.81,A -85,B 0,C 180,E1 9039.474,E2 9039.474} C_VEL
LIN {X 0,Y 417.675,Z 602.81,A -85,B 0,C 180,E1 9050.502,E2 9050.502} C_VEL
LIN {X 0,Y 417.87,Z 602.81,A -85,B 0,C 180,E1 9060.626,E2 9060.626} C_VEL
LIN {X 0,Y 418.155,Z 602.81,A -85,B 0,C 180,E1 9072.017,E2 9072.017} C_VEL
LIN {X 0,Y 418.876,Z 602.81,A -85,B 0,C 180,E1 9082.699,E2 9082.699} C_VEL
LIN {X 0,Y 419.001,Z 602.81,A -85,B 0,C 180,E1 9091.021,E2 9091.021} C_VEL
LIN {X 0,Y 418.622,Z 602.81,A -85,B 0,C 180,E1 9101.482,E2 9101.482} C_VEL
LIN {X 0,Y 418.257,Z 602.81,A -85,B 0,C 180,E1 9112.372,E2 9112.372} C_VEL
LIN {X 0,Y 417.95,Z 602.81,A -85,B 0,C 180,E1 9121.744,E2 9121.744} C_VEL
LIN {X 0,Y 417.854,Z 602.81,A -85,B 0,C 180,E1 9132.183,E2 9132.183} C_VEL
LIN {X 0,Y 417.814,Z 602.81,A -85,B 0,C 180,E1 9143.184,E2 9143.184} C_VEL
LIN {X 0,Y 418.173,Z 604.079,A -85,B 0,C 180,E1 9150.719,E2 9150.719} C_VEL
LIN {X 0,Y 432.109,Z 653.522,A -85,B 0,C 180,E1 9153.26,E2 9153.26} C_VEL
LIN {X 0,Y 427.685,Z 704.964,A -85,B 0,C 180,E1 9156.847,E2 9156.847} C_VEL
LIN {X 0,Y 423.603,Z 745.978,A -85,B 0,C 180,E1 9161.959,E2 9161.959} C_VEL
LIN {X 0,Y 420.52,Z 776.452,A -85,B 0,C 180,E1 9168.554,E2 9168.554} C_VEL
LIN {X 0,Y 419.5,Z 791.188,A -85,B 0,C 180,E1 9174.813,E2 9174.813} C_VEL
LIN {X 0,Y 419.148,Z 794.992,A -85,B 0,C 180,E1 9181.039,E2 9181.039} C_VEL
LIN {X 0,Y 420.077,Z 786.257,A -85,B 0,C 180,E1 9188.31,E2 9188.31} C_VEL
LIN {X 0,Y 422.639,Z 762.501,A -85,B 0,C 180,E1 9195.357,E2 9195.357} C_VEL
LIN {X 0,Y 426.663,Z 725.768,A -85,B 0,C 180,E1 9201.245,E2 9201.245} C_VEL
LIN {X 0,Y 431.322,Z 679.189,A -85,B 0,C 180,E1 9205.531,E2 9205.531} C_VEL
LIN {X 0,Y 431.763,Z 641.043,A -85,B 0,C 180,E1 9207.724,E2 9207.724} C_VEL
LIN {X 0,Y 417.998,Z 602.81,A -85,B 0,C 180,E1 9210.55,E2 9210.55} C_VEL
LIN {X 0,Y 417.862,Z 602.81,A -85,B 0,C 180,E1 9219.46,E2 9219.46} C_VEL
LIN {X 0,Y 417.734,Z 602.81,A -85,B 0,C 180,E1 9230.553,E2 9230.553} C_VEL
LIN {X 0,Y 418.199,Z 604.809,A -85,B 0,C 180,E1 9238.931,E2 9238.931} C_VEL
LIN {X 0,Y 432.717,Z 642.315,A -85,B 0,C 180,E1 9241.373,E2 9241.373} C_VEL
LIN {X 0,Y 430.637,Z 703.724,A -85,B 0,C 180,E1 9243.541,E2 9243.541} C_VEL
LIN {X 0,Y 428.152,Z 732.792,A -85,B 0,C 180,E1 9245.387,E2 9245.387} C_VEL
LIN {X 0,Y 417.808,Z 762.213,A -85,B 0,C 180,E1 9247.681,E2 9247.681} C_VEL
LIN {X 0,Y 413.931,Z 802.99,A -85,B 0,C 180,E1 9253.548,E2 9253.548} C_VEL
LIN {X 0,Y 411.869,Z 830.071,A -85,B 0,C 180,E1 9260.475,E2 9260.475} C_VEL
LIN {X 0,Y 411.581,Z 841.408,A -85,B 0,C 180,E1 9266.847,E2 9266.847} C_VEL
LIN {X 0,Y 411.658,Z 841.508,A -85,B 0,C 180,E1 9273.187,E2 9273.187} C_VEL
LIN {X 0,Y 412.116,Z 827.329,A -85,B 0,C 180,E1 9280.626,E2 9280.626} C_VEL
LIN {X 0,Y 414.19,Z 798.241,A -85,B 0,C 180,E1 9287.452,E2 9287.452} C_VEL
LIN {X 0,Y 418.497,Z 756.714,A -85,B 0,C 180,E1 9292.958,E2 9292.958} C_VEL
LIN {X 0,Y 423.006,Z 705.865,A -85,B 0,C 180,E1 9296.746,E2 9296.746} C_VEL
LIN {X 0,Y 425.451,Z 646.308,A -85,B 0,C 180,E1 9298.691,E2 9298.691} C_VEL
LIN {X 0,Y 410.083,Z 602.81,A -85,B 0,C 180,E1 9300.683,E2 9300.683} C_VEL
LIN {X 0,Y 409.789,Z 602.81,A -85,B 0,C 180,E1 9310.61,E2 9310.61} C_VEL
LIN {X 0,Y 409.724,Z 602.81,A -85,B 0,C 180,E1 9319.596,E2 9319.596} C_VEL
LIN {X 0,Y 409.898,Z 602.81,A -85,B 0,C 180,E1 9330.485,E2 9330.485} C_VEL
LIN {X 0,Y 410.351,Z 604.412,A -85,B 0,C 180,E1 9339.924,E2 9339.924} C_VEL
LIN {X 0,Y 420.419,Z 643.54,A -85,B 0,C 180,E1 9342.877,E2 9342.877} C_VEL
LIN {X 0,Y 417.136,Z 682.306,A -85,B 0,C 180,E1 9346.856,E2 9346.856} C_VEL
LIN {X 0,Y 414.366,Z 706.526,A -85,B 0,C 180,E1 9351.71,E2 9351.71} C_VEL
LIN {X 0,Y 413.137,Z 717.363,A -85,B 0,C 180,E1 9356.84,E2 9356.84} C_VEL
LIN {X 0,Y 412.803,Z 716.515,A -85,B 0,C 180,E1 9362.105,E2 9362.105} C_VEL
LIN {X 0,Y 413.486,Z 701.037,A -85,B 0,C 180,E1 9368,E2 9368} C_VEL
LIN {X 0,Y 415.347,Z 672.01,A -85,B 0,C 180,E1 9372.929,E2 9372.929} C_VEL
LIN {X 0,Y 416.994,Z 630.697,A -85,B 0,C 180,E1 9376.516,E2 9376.516} C_VEL
LIN {X 0,Y 410.516,Z 602.81,A -85,B 0,C 180,E1 9378.311,E2 9378.311} C_VEL
LIN {X 0,Y 409.954,Z 602.81,A -85,B 0,C 180,E1 9389.529,E2 9389.529} C_VEL
LIN {X 0,Y 409.643,Z 602.81,A -85,B 0,C 180,E1 9400.567,E2 9400.567} C_VEL
LIN {X 0,Y 409.622,Z 602.81,A -85,B 0,C 180,E1 9409.567,E2 9409.567} C_VEL
LIN {X 0,Y 409.878,Z 602.81,A -85,B 0,C 180,E1 9420.459,E2 9420.459} C_VEL
LIN {X 0,Y 410.075,Z 602.81,A -85,B 0,C 180,E1 9431.65,E2 9431.65} C_VEL
LIN {X 0,Y 410.848,Z 602.81,A -85,B 0,C 180,E1 9442.556,E2 9442.556} C_VEL
LIN {X 0,Y 411.01,Z 602.81,A -85,B 0,C 180,E1 9451.04,E2 9451.04} C_VEL
LIN {X 0,Y 410.622,Z 602.81,A -85,B 0,C 180,E1 9461.709,E2 9461.709} C_VEL
LIN {X 0,Y 410.19,Z 602.81,A -85,B 0,C 180,E1 9472.837,E2 9472.837} C_VEL
LIN {X 0,Y 409.822,Z 602.81,A -85,B 0,C 180,E1 9483.582,E2 9483.582} C_VEL
LIN {X 0,Y 409.71,Z 602.81,A -85,B 0,C 180,E1 9493.763,E2 9493.763} C_VEL
LIN {X 0,Y 409.761,Z 602.81,A -85,B 0,C 180,E1 9504.971,E2 9504.971} C_VEL
LIN {X 0,Y 410.141,Z 604.412,A -85,B 0,C 180,E1 9510.237,E2 9510.237} C_VEL
LIN {X 0,Y 424.627,Z 654.802,A -85,B 0,C 180,E1 9512.914,E2 9512.914} C_VEL
LIN {X 0,Y 419.993,Z 706.502,A -85,B 0,C 180,E1 9516.624,E2 9516.624} C_VEL
LIN {X 0,Y 415.66,Z 747.69,A -85,B 0,C 180,E1 9521.924,E2 9521.924} C_VEL
LIN {X 0,Y 412.634,Z 776.615,A -85,B 0,C 180,E1 9528.332,E2 9528.332} C_VEL
LIN {X 0,Y 411.549,Z 791.549,A -85,B 0,C 180,E1 9534.713,E2 9534.713} C_VEL
LIN {X 0,Y 411.165,Z 795.482,A -85,B 0,C 180,E1 9541.059,E2 9541.059} C_VEL
LIN {X 0,Y 412.163,Z 786.835,A -85,B 0,C 180,E1 9548.47,E2 9548.47} C_VEL
LIN {X 0,Y 414.898,Z 763.149,A -85,B 0,C 180,E1 9555.65,E2 9555.65} C_VEL
LIN {X 0,Y 419.234,Z 726.541,A -85,B 0,C 180,E1 9561.64,E2 9561.64} C_VEL
LIN {X 0,Y 424.199,Z 680.321,A -85,B 0,C 180,E1 9565.992,E2 9565.992} C_VEL
LIN {X 0,Y 424.921,Z 643.323,A -85,B 0,C 180,E1 9568.203,E2 9568.203} C_VEL
LIN {X 0,Y 409.955,Z 602.81,A -85,B 0,C 180,E1 9571.288,E2 9571.288} C_VEL
LIN {X 0,Y 409.751,Z 602.81,A -85,B 0,C 180,E1 9580.638,E2 9580.638} C_VEL
LIN {X 0,Y 409.653,Z 602.81,A -85,B 0,C 180,E1 9589.617,E2 9589.617} C_VEL
LIN {X 0,Y 410.02,Z 604.542,A -85,B 0,C 180,E1 9597.967,E2 9597.967} C_VEL
LIN {X 0,Y 424.951,Z 640.389,A -85,B 0,C 180,E1 9600.658,E2 9600.658} C_VEL
LIN {X 0,Y 426.16,Z 669.084,A -85,B 0,C 180,E1 9601.603,E2 9601.603} C_VEL
LIN {X 0,Y 421.511,Z 725.331,A -85,B 0,C 180,E1 9604.395,E2 9604.395} C_VEL
LIN {X 0,Y 417.808,Z 762.213,A -85,B 0,C 180,E1 9607.681,E2 9607.681} C_VEL
LIN {X 0,Y 407.172,Z 788.107,A -85,B 0,C 180,E1 9610.706,E2 9610.706} C_VEL
LIN {X 0,Y 404.421,Z 820.03,A -85,B 0,C 180,E1 9617.221,E2 9617.221} C_VEL
LIN {X 0,Y 403.827,Z 838.518,A -85,B 0,C 180,E1 9624.628,E2 9624.628} C_VEL
LIN {X 0,Y 403.661,Z 842.254,A -85,B 0,C 180,E1 9631.095,E2 9631.095} C_VEL
LIN {X 0,Y 403.625,Z 833.65,A -85,B 0,C 180,E1 9638.122,E2 9638.122} C_VEL
LIN {X 0,Y 405.277,Z 810.38,A -85,B 0,C 180,E1 9645.212,E2 9645.212} C_VEL
LIN {X 0,Y 408.918,Z 773.66,A -85,B 0,C 180,E1 9651.322,E2 9651.322} C_VEL
LIN {X 0,Y 413.757,Z 726.143,A -85,B 0,C 180,E1 9655.874,E2 9655.874} C_VEL
LIN {X 0,Y 417.818,Z 672.181,A -85,B 0,C 180,E1 9658.491,E2 9658.491} C_VEL
LIN {X 0,Y 416.033,Z 641.494,A -85,B 0,C 180,E1 9659.355,E2 9659.355} C_VEL
LIN {X 0,Y 401.989,Z 602.81,A -85,B 0,C 180,E1 9661.446,E2 9661.446} C_VEL
LIN {X 0,Y 401.686,Z 602.81,A -85,B 0,C 180,E1 9672.549,E2 9672.549} C_VEL
LIN {X 0,Y 401.629,Z 602.81,A -85,B 0,C 180,E1 9681.432,E2 9681.432} C_VEL
LIN {X 0,Y 401.87,Z 602.81,A -85,B 0,C 180,E1 9692.574,E2 9692.574} C_VEL
LIN {X 0,Y 402.319,Z 604.742,A -85,B 0,C 180,E1 9699.198,E2 9699.198} C_VEL
LIN {X 0,Y 413.274,Z 644.074,A -85,B 0,C 180,E1 9702.384,E2 9702.384} C_VEL
LIN {X 0,Y 409.793,Z 682.439,A -85,B 0,C 180,E1 9706.344,E2 9706.344} C_VEL
LIN {X 0,Y 406.612,Z 708.215,A -85,B 0,C 180,E1 9711.575,E2 9711.575} C_VEL
LIN {X 0,Y 405.281,Z 718.736,A -85,B 0,C 180,E1 9716.779,E2 9716.779} C_VEL
LIN {X 0,Y 404.898,Z 717.64,A -85,B 0,C 180,E1 9722.146,E2 9722.146} C_VEL
LIN {X 0,Y 405.581,Z 702.184,A -85,B 0,C 180,E1 9728.064,E2 9728.064} C_VEL
LIN {X 0,Y 407.555,Z 672.293,A -85,B 0,C 180,E1 9733.181,E2 9733.181} C_VEL
LIN {X 0,Y 409.168,Z 632.026,A -85,B 0,C 180,E1 9736.732,E2 9736.732} C_VEL
LIN {X 0,Y 402.524,Z 602.81,A -85,B 0,C 180,E1 9738.457,E2 9738.457} C_VEL
LIN {X 0,Y 401.924,Z 602.81,A -85,B 0,C 180,E1 9748.158,E2 9748.158} C_VEL
LIN {X 0,Y 401.539,Z 602.81,A -85,B 0,C 180,E1 9759.197,E2 9759.197} C_VEL
LIN {X 0,Y 401.542,Z 602.81,A -85,B 0,C 180,E1 9768.578,E2 9768.578} C_VEL
LIN {X 0,Y 401.709,Z 602.81,A -85,B 0,C 180,E1 9779.32,E2 9779.32} C_VEL
LIN {X 0,Y 401.839,Z 602.81,A -85,B 0,C 180,E1 9788.959,E2 9788.959} C_VEL
LIN {X 0,Y 402.677,Z 602.81,A -85,B 0,C 180,E1 9800.219,E2 9800.219} C_VEL
LIN {X 0,Y 403.004,Z 602.81,A -85,B 0,C 180,E1 9811.061,E2 9811.061} C_VEL
LIN {X 0,Y 402.584,Z 602.81,A -85,B 0,C 180,E1 9821.946,E2 9821.946} C_VEL
LIN {X 0,Y 402.155,Z 602.81,A -85,B 0,C 180,E1 9833.32,E2 9833.32} C_VEL
LIN {X 0,Y 401.812,Z 602.81,A -85,B 0,C 180,E1 9843.179,E2 9843.179} C_VEL
LIN {X 0,Y 401.642,Z 602.81,A -85,B 0,C 180,E1 9854.315,E2 9854.315} C_VEL
LIN {X 0,Y 401.724,Z 602.81,A -85,B 0,C 180,E1 9864.269,E2 9864.269} C_VEL
LIN {X 0,Y 402.122,Z 604.737,A -85,B 0,C 180,E1 9869.738,E2 9869.738} C_VEL
LIN {X 0,Y 417.188,Z 655.511,A -85,B 0,C 180,E1 9872.535,E2 9872.535} C_VEL
LIN {X 0,Y 412.369,Z 707.095,A -85,B 0,C 180,E1 9876.311,E2 9876.311} C_VEL
LIN {X 0,Y 407.732,Z 749.088,A -85,B 0,C 180,E1 9881.84,E2 9881.84} C_VEL
LIN {X 0,Y 404.546,Z 778.534,A -85,B 0,C 180,E1 9888.644,E2 9888.644} C_VEL
LIN {X 0,Y 403.543,Z 792.982,A -85,B 0,C 180,E1 9895.427,E2 9895.427} C_VEL
LIN {X 0,Y 403.183,Z 795.978,A -85,B 0,C 180,E1 9901.08,E2 9901.08} C_VEL
LIN {X 0,Y 404.283,Z 787.438,A -85,B 0,C 180,E1 9908.637,E2 9908.637} C_VEL
LIN {X 0,Y 407.024,Z 765.045,A -85,B 0,C 180,E1 9915.684,E2 9915.684} C_VEL
LIN {X 0,Y 411.563,Z 729.483,A -85,B 0,C 180,E1 9921.78,E2 9921.78} C_VEL
LIN {X 0,Y 416.988,Z 683.433,A -85,B 0,C 180,E1 9926.33,E2 9926.33} C_VEL
LIN {X 0,Y 418.202,Z 645.649,A -85,B 0,C 180,E1 9928.705,E2 9928.705} C_VEL
LIN {X 0,Y 404.04,Z 608.251,A -85,B 0,C 180,E1 9931.779,E2 9931.779} C_VEL
LIN {X 0,Y 401.823,Z 602.81,A -85,B 0,C 180,E1 9932.496,E2 9932.496} C_VEL
LIN {X 0,Y 401.627,Z 602.81,A -85,B 0,C 180,E1 9942.574,E2 9942.574} C_VEL
LIN {X 0,Y 401.685,Z 602.81,A -85,B 0,C 180,E1 9954.183,E2 9954.183} C_VEL
LIN {X 0,Y 401.959,Z 604.72,A -85,B 0,C 180,E1 9956.905,E2 9956.905} C_VEL
LIN {X 0,Y 417.908,Z 640.623,A -85,B 0,C 180,E1 9960.007,E2 9960.007} C_VEL
LIN {X 0,Y 419.484,Z 666.438,A -85,B 0,C 180,E1 9960.951,E2 9960.951} C_VEL
LIN {X 0,Y 414.494,Z 723.12,A -85,B 0,C 180,E1 9963.764,E2 9963.764} C_VEL
LIN {X 0,Y 409.017,Z 772.617,A -85,B 0,C 180,E1 9968.524,E2 9968.524} C_VEL
LIN {X 0,Y 407.172,Z 788.107,A -85,B 0,C 180,E1 9970.706,E2 9970.706} C_VEL
LIN {X 0,Y 397.299,Z 809.753,A -85,B 0,C 180,E1 9974.483,E2 9974.483} C_VEL
LIN {X 0,Y 395.679,Z 833.153,A -85,B 0,C 180,E1 9981.75,E2 9981.75} C_VEL
LIN {X 0,Y 395.901,Z 841.74,A -85,B 0,C 180,E1 9988.92,E2 9988.92} C_VEL
LIN {X 0,Y 395.687,Z 837.984,A -85,B 0,C 180,E1 9995.519,E2 9995.519} C_VEL
LIN {X 0,Y 396.196,Z 820.777,A -85,B 0,C 180,E1 10002.683,E2 10002.683} C_VEL
LIN {X 0,Y 399.026,Z 790.335,A -85,B 0,C 180,E1 10009.165,E2 10009.165} C_VEL
LIN {X 0,Y 404.044,Z 746.573,A -85,B 0,C 180,E1 10014.567,E2 10014.567} C_VEL
LIN {X 0,Y 409.086,Z 693.331,A -85,B 0,C 180,E1 10018.128,E2 10018.128} C_VEL
LIN {X 0,Y 409.177,Z 644.833,A -85,B 0,C 180,E1 10019.692,E2 10019.692} C_VEL
LIN {X 0,Y 393.872,Z 602.81,A -85,B 0,C 180,E1 10022.336,E2 10022.336} C_VEL
LIN {X 0,Y 393.68,Z 602.81,A -85,B 0,C 180,E1 10032.44,E2 10032.44} C_VEL
LIN {X 0,Y 393.566,Z 602.81,A -85,B 0,C 180,E1 10043.297,E2 10043.297} C_VEL
LIN {X 0,Y 393.867,Z 602.81,A -85,B 0,C 180,E1 10053.698,E2 10053.698} C_VEL
LIN {X 0,Y 394.191,Z 604.476,A -85,B 0,C 180,E1 10058.356,E2 10058.356} C_VEL
LIN {X 0,Y 405.876,Z 643.195,A -85,B 0,C 180,E1 10061.712,E2 10061.712} C_VEL
LIN {X 0,Y 402.495,Z 682.771,A -85,B 0,C 180,E1 10065.813,E2 10065.813} C_VEL
LIN {X 0,Y 398.992,Z 708.873,A -85,B 0,C 180,E1 10071.096,E2 10071.096} C_VEL
LIN {X 0,Y 397.41,Z 720.117,A -85,B 0,C 180,E1 10076.715,E2 10076.715} C_VEL
LIN {X 0,Y 397.012,Z 718.749,A -85,B 0,C 180,E1 10082.189,E2 10082.189} C_VEL
LIN {X 0,Y 397.716,Z 702.938,A -85,B 0,C 180,E1 10088.224,E2 10088.224} C_VEL
LIN {X 0,Y 399.78,Z 672.557,A -85,B 0,C 180,E1 10093.442,E2 10093.442} C_VEL
LIN {X 0,Y 401.053,Z 631.587,A -85,B 0,C 180,E1 10097.081,E2 10097.081} C_VEL
LIN {X 0,Y 394.477,Z 602.81,A -85,B 0,C 180,E1 10098.8,E2 10098.8} C_VEL
LIN {X 0,Y 393.745,Z 602.81,A -85,B 0,C 180,E1 10109.844,E2 10109.844} C_VEL
LIN {X 0,Y 393.532,Z 602.81,A -85,B 0,C 180,E1 10121.22,E2 10121.22} C_VEL
LIN {X 0,Y 393.454,Z 602.81,A -85,B 0,C 180,E1 10132.243,E2 10132.243} C_VEL
LIN {X 0,Y 393.812,Z 602.81,A -85,B 0,C 180,E1 10143.678,E2 10143.678} C_VEL
LIN {X 0,Y 394.245,Z 602.81,A -85,B 0,C 180,E1 10155.494,E2 10155.494} C_VEL
LIN {X 0,Y 395.006,Z 602.81,A -85,B 0,C 180,E1 10166.679,E2 10166.679} C_VEL
LIN {X 0,Y 394.871,Z 602.81,A -85,B 0,C 180,E1 10177.711,E2 10177.711} C_VEL
LIN {X 0,Y 394.254,Z 602.81,A -85,B 0,C 180,E1 10189.076,E2 10189.076} C_VEL
LIN {X 0,Y 393.81,Z 602.81,A -85,B 0,C 180,E1 10199.892,E2 10199.892} C_VEL
LIN {X 0,Y 393.698,Z 602.81,A -85,B 0,C 180,E1 10211.272,E2 10211.272} C_VEL
LIN {X 0,Y 393.601,Z 602.81,A -85,B 0,C 180,E1 10222.183,E2 10222.183} C_VEL
LIN {X 0,Y 393.779,Z 603.07,A -85,B 0,C 180,E1 10229.16,E2 10229.16} C_VEL
LIN {X 0,Y 409.722,Z 656.304,A -85,B 0,C 180,E1 10232.154,E2 10232.154} C_VEL
LIN {X 0,Y 404.772,Z 707.171,A -85,B 0,C 180,E1 10235.941,E2 10235.941} C_VEL
LIN {X 0,Y 400.012,Z 748.977,A -85,B 0,C 180,E1 10241.505,E2 10241.505} C_VEL
LIN {X 0,Y 396.649,Z 778.658,A -85,B 0,C 180,E1 10248.415,E2 10248.415} C_VEL
LIN {X 0,Y 395.558,Z 793.352,A -85,B 0,C 180,E1 10255.334,E2 10255.334} C_VEL
LIN {X 0,Y 395.221,Z 796.476,A -85,B 0,C 180,E1 10261.102,E2 10261.102} C_VEL
LIN {X 0,Y 396.382,Z 788.073,A -85,B 0,C 180,E1 10268.81,E2 10268.81} C_VEL
LIN {X 0,Y 399.472,Z 764.63,A -85,B 0,C 180,E1 10276.271,E2 10276.271} C_VEL
LIN {X 0,Y 404.509,Z 728.432,A -85,B 0,C 180,E1 10282.47,E2 10282.47} C_VEL
LIN {X 0,Y 410.364,Z 681.468,A -85,B 0,C 180,E1 10287.086,E2 10287.086} C_VEL
LIN {X 0,Y 411.322,Z 646.72,A -85,B 0,C 180,E1 10289.332,E2 10289.332} C_VEL
LIN {X 0,Y 397.815,Z 611.778,A -85,B 0,C 180,E1 10292.497,E2 10292.497} C_VEL
LIN {X 0,Y 393.719,Z 602.81,A -85,B 0,C 180,E1 10293.659,E2 10293.659} C_VEL
LIN {X 0,Y 393.606,Z 602.81,A -85,B 0,C 180,E1 10304.532,E2 10304.532} C_VEL
LIN {X 0,Y 393.939,Z 604.615,A -85,B 0,C 180,E1 10315.675,E2 10315.675} C_VEL
LIN {X 0,Y 411.003,Z 641.018,A -85,B 0,C 180,E1 10319.315,E2 10319.315} C_VEL
LIN {X 0,Y 412.964,Z 664.433,A -85,B 0,C 180,E1 10320.282,E2 10320.282} C_VEL
LIN {X 0,Y 407.435,Z 722.228,A -85,B 0,C 180,E1 10323.185,E2 10323.185} C_VEL
LIN {X 0,Y 401.48,Z 772.29,A -85,B 0,C 180,E1 10328.097,E2 10328.097} C_VEL
LIN {X 0,Y 397.299,Z 809.753,A -85,B 0,C 180,E1 10334.483,E2 10334.483} C_VEL
LIN {X 0,Y 388.288,Z 826.101,A -85,B 0,C 180,E1 10338.892,E2 10338.892} C_VEL
LIN {X 0,Y 387.652,Z 840.055,A -85,B 0,C 180,E1 10346.652,E2 10346.652} C_VEL
LIN {X 0,Y 387.694,Z 839.859,A -85,B 0,C 180,E1 10353.506,E2 10353.506} C_VEL
LIN {X 0,Y 388.116,Z 825.214,A -85,B 0,C 180,E1 10361.29,E2 10361.29} C_VEL
LIN {X 0,Y 390.509,Z 796.945,A -85,B 0,C 180,E1 10368.202,E2 10368.202} C_VEL
LIN {X 0,Y 395.529,Z 754.695,A -85,B 0,C 180,E1 10374.074,E2 10374.074} C_VEL
LIN {X 0,Y 400.782,Z 703.3,A -85,B 0,C 180,E1 10378.043,E2 10378.043} C_VEL
LIN {X 0,Y 402.368,Z 647.204,A -85,B 0,C 180,E1 10380.191,E2 10380.191} C_VEL
LIN {X 0,Y 386.577,Z 606.153,A -85,B 0,C 180,E1 10383.018,E2 10383.018} C_VEL
LIN {X 0,Y 385.799,Z 602.81,A -85,B 0,C 180,E1 10383.489,E2 10383.489} C_VEL
LIN {X 0,Y 385.612,Z 602.81,A -85,B 0,C 180,E1 10393.546,E2 10393.546} C_VEL
LIN {X 0,Y 385.549,Z 602.81,A -85,B 0,C 180,E1 10405.199,E2 10405.199} C_VEL
LIN {X 0,Y 385.949,Z 602.81,A -85,B 0,C 180,E1 10416.631,E2 10416.631} C_VEL
LIN {X 0,Y 386.389,Z 605.273,A -85,B 0,C 180,E1 10417.501,E2 10417.501} C_VEL
LIN {X 0,Y 398.271,Z 641.841,A -85,B 0,C 180,E1 10420.929,E2 10420.929} C_VEL
LIN {X 0,Y 395.411,Z 681.228,A -85,B 0,C 180,E1 10424.985,E2 10424.985} C_VEL
LIN {X 0,Y 391.756,Z 707.33,A -85,B 0,C 180,E1 10429.96,E2 10429.96} C_VEL
LIN {X 0,Y 389.651,Z 720.466,A -85,B 0,C 180,E1 10435.531,E2 10435.531} C_VEL
LIN {X 0,Y 388.904,Z 721.137,A -85,B 0,C 180,E1 10441.116,E2 10441.116} C_VEL
LIN {X 0,Y 389.429,Z 707.779,A -85,B 0,C 180,E1 10447.299,E2 10447.299} C_VEL
LIN {X 0,Y 391.279,Z 681.105,A -85,B 0,C 180,E1 10452.599,E2 10452.599} C_VEL
LIN {X 0,Y 393.919,Z 641.431,A -85,B 0,C 180,E1 10456.699,E2 10456.699} C_VEL
LIN {X 0,Y 386.424,Z 602.81,A -85,B 0,C 180,E1 10459.043,E2 10459.043} C_VEL
LIN {X 0,Y 385.757,Z 602.81,A -85,B 0,C 180,E1 10469.452,E2 10469.452} C_VEL
LIN {X 0,Y 385.495,Z 602.81,A -85,B 0,C 180,E1 10480.502,E2 10480.502} C_VEL
LIN {X 0,Y 385.483,Z 602.81,A -85,B 0,C 180,E1 10490.139,E2 10490.139} C_VEL
LIN {X 0,Y 385.68,Z 602.81,A -85,B 0,C 180,E1 10500.521,E2 10500.521} C_VEL
LIN {X 0,Y 385.895,Z 602.81,A -85,B 0,C 180,E1 10510.455,E2 10510.455} C_VEL
LIN {X 0,Y 386.753,Z 602.81,A -85,B 0,C 180,E1 10522.089,E2 10522.089} C_VEL
LIN {X 0,Y 387.016,Z 602.81,A -85,B 0,C 180,E1 10531.105,E2 10531.105} C_VEL
LIN {X 0,Y 386.523,Z 602.81,A -85,B 0,C 180,E1 10542.45,E2 10542.45} C_VEL
LIN {X 0,Y 386.064,Z 602.81,A -85,B 0,C 180,E1 10552.532,E2 10552.532} C_VEL
LIN {X 0,Y 385.704,Z 602.81,A -85,B 0,C 180,E1 10562.238,E2 10562.238} C_VEL
LIN {X 0,Y 385.606,Z 602.81,A -85,B 0,C 180,E1 10573.496,E2 10573.496} C_VEL
LIN {X 0,Y 385.547,Z 602.81,A -85,B 0,C 180,E1 10583.753,E2 10583.753} C_VEL
LIN {X 0,Y 385.975,Z 604.816,A -85,B 0,C 180,E1 10588.691,E2 10588.691} C_VEL
LIN {X 0,Y 402.212,Z 657.547,A -85,B 0,C 180,E1 10591.788,E2 10591.788} C_VEL
LIN {X 0,Y 397.023,Z 709.004,A -85,B 0,C 180,E1 10595.742,E2 10595.742} C_VEL
LIN {X 0,Y 392.099,Z 750.239,A -85,B 0,C 180,E1 10601.405,E2 10601.405} C_VEL
LIN {X 0,Y 388.756,Z 778.74,A -85,B 0,C 180,E1 10608.176,E2 10608.176} C_VEL
LIN {X 0,Y 387.574,Z 794.16,A -85,B 0,C 180,E1 10615.623,E2 10615.623} C_VEL
LIN {X 0,Y 387.702,Z 796.093,A -85,B 0,C 180,E1 10623.368,E2 10623.368} C_VEL
LIN {X 0,Y 389.068,Z 783.612,A -85,B 0,C 180,E1 10631.247,E2 10631.247} C_VEL
LIN {X 0,Y 392.749,Z 757.392,A -85,B 0,C 180,E1 10638.375,E2 10638.375} C_VEL
LIN {X 0,Y 398.961,Z 717.488,A -85,B 0,C 180,E1 10644.398,E2 10644.398} C_VEL
LIN {X 0,Y 405.317,Z 666.646,A -85,B 0,C 180,E1 10648.717,E2 10648.717} C_VEL
LIN {X 0,Y 402.468,Z 639.173,A -85,B 0,C 180,E1 10650.707,E2 10650.707} C_VEL
LIN {X 0,Y 387.289,Z 607.623,A -85,B 0,C 180,E1 10654.401,E2 10654.401} C_VEL
LIN {X 0,Y 385.587,Z 602.81,A -85,B 0,C 180,E1 10655.529,E2 10655.529} C_VEL
LIN {X 0,Y 385.528,Z 602.81,A -85,B 0,C 180,E1 10666.736,E2 10666.736} C_VEL
LIN {X 0,Y 385.853,Z 604.764,A -85,B 0,C 180,E1 10674.211,E2 10674.211} C_VEL
LIN {X 0,Y 403.009,Z 638.55,A -85,B 0,C 180,E1 10678.326,E2 10678.326} C_VEL
LIN {X 0,Y 406.64,Z 661.625,A -85,B 0,C 180,E1 10679.54,E2 10679.54} C_VEL
LIN {X 0,Y 400.605,Z 720.029,A -85,B 0,C 180,E1 10682.473,E2 10682.473} C_VEL
LIN {X 0,Y 394.201,Z 770.522,A -85,B 0,C 180,E1 10687.451,E2 10687.451} C_VEL
LIN {X 0,Y 389.662,Z 808.284,A -85,B 0,C 180,E1 10693.911,E2 10693.911} C_VEL
LIN {X 0,Y 388.288,Z 826.101,A -85,B 0,C 180,E1 10698.892,E2 10698.892} C_VEL
LIN {X 0,Y 379.796,Z 836.462,A -85,B 0,C 180,E1 10703.801,E2 10703.801} C_VEL
LIN {X 0,Y 379.718,Z 840.741,A -85,B 0,C 180,E1 10711.164,E2 10711.164} C_VEL
LIN {X 0,Y 379.838,Z 831.707,A -85,B 0,C 180,E1 10718.634,E2 10718.634} C_VEL
LIN {X 0,Y 381.762,Z 807.562,A -85,B 0,C 180,E1 10726.174,E2 10726.174} C_VEL
LIN {X 0,Y 385.912,Z 770.818,A -85,B 0,C 180,E1 10732.468,E2 10732.468} C_VEL
LIN {X 0,Y 391.504,Z 721.848,A -85,B 0,C 180,E1 10737.274,E2 10737.274} C_VEL
LIN {X 0,Y 397.016,Z 656.416,A -85,B 0,C 180,E1 10740.426,E2 10740.426} C_VEL
LIN {X 0,Y 381.962,Z 612.349,A -85,B 0,C 180,E1 10743.393,E2 10743.393} C_VEL
LIN {X 0,Y 377.714,Z 602.81,A -85,B 0,C 180,E1 10744.551,E2 10744.551} C_VEL
LIN {X 0,Y 377.483,Z 602.81,A -85,B 0,C 180,E1 10755.289,E2 10755.289} C_VEL
LIN {X 0,Y 377.553,Z 602.81,A -85,B 0,C 180,E1 10767.137,E2 10767.137} C_VEL
LIN {X 0,Y 378.124,Z 604.533,A -85,B 0,C 180,E1 10776.404,E2 10776.404} C_VEL
LIN {X 0,Y 391.036,Z 642.074,A -85,B 0,C 180,E1 10780.255,E2 10780.255} C_VEL
LIN {X 0,Y 388.275,Z 681.695,A -85,B 0,C 180,E1 10784.412,E2 10784.412} C_VEL
LIN {X 0,Y 384.107,Z 709.188,A -85,B 0,C 180,E1 10789.758,E2 10789.758} C_VEL
LIN {X 0,Y 381.826,Z 721.928,A -85,B 0,C 180,E1 10795.439,E2 10795.439} C_VEL
LIN {X 0,Y 381.016,Z 722.296,A -85,B 0,C 180,E1 10801.139,E2 10801.139} C_VEL
LIN {X 0,Y 381.471,Z 709.563,A -85,B 0,C 180,E1 10807.151,E2 10807.151} C_VEL
LIN {X 0,Y 383.328,Z 683.302,A -85,B 0,C 180,E1 10812.574,E2 10812.574} C_VEL
LIN {X 0,Y 386.062,Z 643.91,A -85,B 0,C 180,E1 10816.82,E2 10816.82} C_VEL
LIN {X 0,Y 378.382,Z 602.81,A -85,B 0,C 180,E1 10819.489,E2 10819.489} C_VEL
LIN {X 0,Y 377.641,Z 602.81,A -85,B 0,C 180,E1 10830.209,E2 10830.209} C_VEL
LIN {X 0,Y 377.401,Z 602.81,A -85,B 0,C 180,E1 10841.916,E2 10841.916} C_VEL
LIN {X 0,Y 377.427,Z 602.81,A -85,B 0,C 180,E1 10851.627,E2 10851.627} C_VEL
LIN {X 0,Y 377.676,Z 602.81,A -85,B 0,C 180,E1 10862.461,E2 10862.461} C_VEL
LIN {X 0,Y 378.17,Z 602.81,A -85,B 0,C 180,E1 10874.863,E2 10874.863} C_VEL
LIN {X 0,Y 378.983,Z 602.81,A -85,B 0,C 180,E1 10886.538,E2 10886.538} C_VEL
LIN {X 0,Y 378.79,Z 602.81,A -85,B 0,C 180,E1 10898.041,E2 10898.041} C_VEL
LIN {X 0,Y 378.175,Z 602.81,A -85,B 0,C 180,E1 10909.921,E2 10909.921} C_VEL
LIN {X 0,Y 377.717,Z 602.81,A -85,B 0,C 180,E1 10920.262,E2 10920.262} C_VEL
LIN {X 0,Y 377.527,Z 602.81,A -85,B 0,C 180,E1 10931.963,E2 10931.963} C_VEL
LIN {X 0,Y 377.536,Z 602.81,A -85,B 0,C 180,E1 10941.573,E2 10941.573} C_VEL
LIN {X 0,Y 377.664,Z 603.145,A -85,B 0,C 180,E1 10948.09,E2 10948.09} C_VEL
LIN {X 0,Y 394.695,Z 659.036,A -85,B 0,C 180,E1 10951.431,E2 10951.431} C_VEL
LIN {X 0,Y 389.236,Z 710.642,A -85,B 0,C 180,E1 10955.531,E2 10955.531} C_VEL
LIN {X 0,Y 384.196,Z 751.229,A -85,B 0,C 180,E1 10961.267,E2 10961.267} C_VEL
LIN {X 0,Y 380.648,Z 780.514,A -85,B 0,C 180,E1 10968.504,E2 10968.504} C_VEL
LIN {X 0,Y 379.593,Z 794.38,A -85,B 0,C 180,E1 10975.416,E2 10975.416} C_VEL
LIN {X 0,Y 379.744,Z 796.665,A -85,B 0,C 180,E1 10983.438,E2 10983.438} C_VEL
LIN {X 0,Y 381.229,Z 784.372,A -85,B 0,C 180,E1 10991.482,E2 10991.482} C_VEL
LIN {X 0,Y 385.297,Z 757.606,A -85,B 0,C 180,E1 10998.909,E2 10998.909} C_VEL
LIN {X 0,Y 391.979,Z 717.567,A -85,B 0,C 180,E1 11005.037,E2 11005.037} C_VEL
LIN {X 0,Y 398.895,Z 666.651,A -85,B 0,C 180,E1 11009.417,E2 11009.417} C_VEL
LIN {X 0,Y 394.514,Z 636.758,A -85,B 0,C 180,E1 11011.849,E2 11011.849} C_VEL
LIN {X 0,Y 379.649,Z 608.119,A -85,B 0,C 180,E1 11015.944,E2 11015.944} C_VEL
LIN {X 0,Y 377.64,Z 602.81,A -85,B 0,C 180,E1 11017.19,E2 11017.19} C_VEL
LIN {X 0,Y 377.404,Z 602.81,A -85,B 0,C 180,E1 11028.467,E2 11028.467} C_VEL
LIN {X 0,Y 377.783,Z 604.825,A -85,B 0,C 180,E1 11032.382,E2 11032.382} C_VEL
LIN {X 0,Y 392.436,Z 630.976,A -85,B 0,C 180,E1 11036.618,E2 11036.618} C_VEL
LIN {X 0,Y 400.579,Z 657.823,A -85,B 0,C 180,E1 11038.73,E2 11038.73} C_VEL
LIN {X 0,Y 394.055,Z 716.872,A -85,B 0,C 180,E1 11041.646,E2 11041.646} C_VEL
LIN {X 0,Y 387.301,Z 766.551,A -85,B 0,C 180,E1 11046.484,E2 11046.484} C_VEL
LIN {X 0,Y 382.272,Z 805.389,A -85,B 0,C 180,E1 11052.998,E2 11052.998} C_VEL
LIN {X 0,Y 379.928,Z 829.783,A -85,B 0,C 180,E1 11060.246,E2 11060.246} C_VEL
LIN {X 0,Y 379.796,Z 836.462,A -85,B 0,C 180,E1 11063.801,E2 11063.801} C_VEL
LIN {X 0,Y 371.88,Z 840.356,A -85,B 0,C 180,E1 11069.045,E2 11069.045} C_VEL
LIN {X 0,Y 371.674,Z 836.174,A -85,B 0,C 180,E1 11075.877,E2 11075.877} C_VEL
LIN {X 0,Y 372.472,Z 817.979,A -85,B 0,C 180,E1 11083.566,E2 11083.566} C_VEL
LIN {X 0,Y 375.873,Z 786.597,A -85,B 0,C 180,E1 11090.396,E2 11090.396} C_VEL
LIN {X 0,Y 381.515,Z 742.267,A -85,B 0,C 180,E1 11095.961,E2 11095.961} C_VEL
LIN {X 0,Y 388.696,Z 678.284,A -85,B 0,C 180,E1 11100.256,E2 11100.256} C_VEL
LIN {X 0,Y 388.463,Z 649.909,A -85,B 0,C 180,E1 11101.467,E2 11101.467} C_VEL
LIN {X 0,Y 374.883,Z 613.709,A -85,B 0,C 180,E1 11104.308,E2 11104.308} C_VEL
LIN {X 0,Y 369.607,Z 602.81,A -85,B 0,C 180,E1 11105.888,E2 11105.888} C_VEL
LIN {X 0,Y 369.421,Z 602.81,A -85,B 0,C 180,E1 11117.328,E2 11117.328} C_VEL
LIN {X 0,Y 369.551,Z 602.81,A -85,B 0,C 180,E1 11129.115,E2 11129.115} C_VEL
LIN {X 0,Y 370.034,Z 604.574,A -85,B 0,C 180,E1 11135.215,E2 11135.215} C_VEL
LIN {X 0,Y 383.685,Z 641.023,A -85,B 0,C 180,E1 11139.389,E2 11139.389} C_VEL
LIN {X 0,Y 382.211,Z 674.801,A -85,B 0,C 180,E1 11142.823,E2 11142.823} C_VEL
LIN {X 0,Y 377.627,Z 705.679,A -85,B 0,C 180,E1 11148.113,E2 11148.113} C_VEL
LIN {X 0,Y 374.584,Z 721.955,A -85,B 0,C 180,E1 11154.185,E2 11154.185} C_VEL
LIN {X 0,Y 373.9,Z 724.745,A -85,B 0,C 180,E1 11158.835,E2 11158.835} C_VEL
LIN {X 0,Y 373.533,Z 715.863,A -85,B 0,C 180,E1 11165.398,E2 11165.398} C_VEL
LIN {X 0,Y 374.956,Z 692.418,A -85,B 0,C 180,E1 11171.377,E2 11171.377} C_VEL
LIN {X 0,Y 377.638,Z 655.221,A -85,B 0,C 180,E1 11176.185,E2 11176.185} C_VEL
LIN {X 0,Y 375.877,Z 626.923,A -85,B 0,C 180,E1 11178.379,E2 11178.379} C_VEL
LIN {X 0,Y 370.294,Z 602.81,A -85,B 0,C 180,E1 11179.932,E2 11179.932} C_VEL
LIN {X 0,Y 369.553,Z 602.81,A -85,B 0,C 180,E1 11190.88,E2 11190.88} C_VEL
LIN {X 0,Y 369.321,Z 602.81,A -85,B 0,C 180,E1 11202.682,E2 11202.682} C_VEL
LIN {X 0,Y 369.346,Z 602.81,A -85,B 0,C 180,E1 11213.414,E2 11213.414} C_VEL
LIN {X 0,Y 369.623,Z 602.81,A -85,B 0,C 180,E1 11224.445,E2 11224.445} C_VEL
LIN {X 0,Y 370.119,Z 602.81,A -85,B 0,C 180,E1 11234.525,E2 11234.525} C_VEL
LIN {X 0,Y 370.978,Z 602.81,A -85,B 0,C 180,E1 11246.463,E2 11246.463} C_VEL
LIN {X 0,Y 370.776,Z 602.81,A -85,B 0,C 180,E1 11258.216,E2 11258.216} C_VEL
LIN {X 0,Y 370.107,Z 602.81,A -85,B 0,C 180,E1 11270.374,E2 11270.374} C_VEL
LIN {X 0,Y 369.647,Z 602.81,A -85,B 0,C 180,E1 11280.849,E2 11280.849} C_VEL
LIN {X 0,Y 369.452,Z 602.81,A -85,B 0,C 180,E1 11292.635,E2 11292.635} C_VEL
LIN {X 0,Y 369.441,Z 602.81,A -85,B 0,C 180,E1 11303.448,E2 11303.448} C_VEL
LIN {X 0,Y 369.789,Z 604.494,A -85,B 0,C 180,E1 11307.58,E2 11307.58} C_VEL
LIN {X 0,Y 387.201,Z 660.073,A -85,B 0,C 180,E1 11311.045,E2 11311.045} C_VEL
LIN {X 0,Y 381.454,Z 712.175,A -85,B 0,C 180,E1 11315.312,E2 11315.312} C_VEL
LIN {X 0,Y 376.035,Z 753.753,A -85,B 0,C 180,E1 11321.429,E2 11321.429} C_VEL
LIN {X 0,Y 372.554,Z 782.205,A -85,B 0,C 180,E1 11328.846,E2 11328.846} C_VEL
LIN {X 0,Y 371.669,Z 795.98,A -85,B 0,C 180,E1 11336.491,E2 11336.491} C_VEL
LIN {X 0,Y 371.775,Z 797.25,A -85,B 0,C 180,E1 11343.512,E2 11343.512} C_VEL
LIN {X 0,Y 373.371,Z 785.18,A -85,B 0,C 180,E1 11351.727,E2 11351.727} C_VEL
LIN {X 0,Y 377.852,Z 758.342,A -85,B 0,C 180,E1 11359.374,E2 11359.374} C_VEL
LIN {X 0,Y 385.116,Z 717.901,A -85,B 0,C 180,E1 11365.688,E2 11365.688} C_VEL
LIN {X 0,Y 392.652,Z 666.601,A -85,B 0,C 180,E1 11370.162,E2 11370.162} C_VEL
LIN {X 0,Y 387.437,Z 636.778,A -85,B 0,C 180,E1 11372.888,E2 11372.888} C_VEL
LIN {X 0,Y 373.342,Z 609.562,A -85,B 0,C 180,E1 11377.473,E2 11377.473} C_VEL
LIN {X 0,Y 369.456,Z 602.81,A -85,B 0,C 180,E1 11379.544,E2 11379.544} C_VEL
LIN {X 0,Y 369.56,Z 604.817,A -85,B 0,C 180,E1 11389.753,E2 11389.753} C_VEL
LIN {X 0,Y 380.779,Z 622.378,A -85,B 0,C 180,E1 11394.183,E2 11394.183} C_VEL
LIN {X 0,Y 393.634,Z 653.614,A -85,B 0,C 180,E1 11397.709,E2 11397.709} C_VEL
LIN {X 0,Y 387.527,Z 715.107,A -85,B 0,C 180,E1 11400.877,E2 11400.877} C_VEL
LIN {X 0,Y 380.022,Z 766.004,A -85,B 0,C 180,E1 11405.909,E2 11405.909} C_VEL
LIN {X 0,Y 374.481,Z 805.165,A -85,B 0,C 180,E1 11412.633,E2 11412.633} C_VEL
LIN {X 0,Y 371.991,Z 829.411,A -85,B 0,C 180,E1 11420.036,E2 11420.036} C_VEL
LIN {X 0,Y 371.692,Z 839.183,A -85,B 0,C 180,E1 11426.508,E2 11426.508} C_VEL
LIN {X 0,Y 371.88,Z 840.356,A -85,B 0,C 180,E1 11429.045,E2 11429.045} C_VEL
LIN {X 0,Y 363.72,Z 837.483,A -85,B 0,C 180,E1 11434.404,E2 11434.404} C_VEL
LIN {X 0,Y 364.225,Z 821.785,A -85,B 0,C 180,E1 11442.368,E2 11442.368} C_VEL
LIN {X 0,Y 367.257,Z 792.067,A -85,B 0,C 180,E1 11449.635,E2 11449.635} C_VEL
LIN {X 0,Y 372.942,Z 749.524,A -85,B 0,C 180,E1 11455.573,E2 11455.573} C_VEL
LIN {X 0,Y 380.999,Z 686.77,A -85,B 0,C 180,E1 11460.481,E2 11460.481} C_VEL
LIN {X 0,Y 382.11,Z 652.608,A -85,B 0,C 180,E1 11462.07,E2 11462.07} C_VEL
LIN {X 0,Y 369.587,Z 618.483,A -85,B 0,C 180,E1 11464.915,E2 11464.915} C_VEL
LIN {X 0,Y 361.474,Z 602.81,A -85,B 0,C 180,E1 11467.216,E2 11467.216} C_VEL
LIN {X 0,Y 361.42,Z 602.81,A -85,B 0,C 180,E1 11477.311,E2 11477.311} C_VEL
LIN {X 0,Y 361.521,Z 602.81,A -85,B 0,C 180,E1 11489.402,E2 11489.402} C_VEL
LIN {X 0,Y 361.965,Z 604.87,A -85,B 0,C 180,E1 11493.853,E2 11493.853} C_VEL
LIN {X 0,Y 376.428,Z 639.994,A -85,B 0,C 180,E1 11498.449,E2 11498.449} C_VEL
LIN {X 0,Y 376.448,Z 668.345,A -85,B 0,C 180,E1 11501.361,E2 11501.361} C_VEL
LIN {X 0,Y 371.383,Z 701.44,A -85,B 0,C 180,E1 11506.41,E2 11506.41} C_VEL
LIN {X 0,Y 367.608,Z 720.426,A -85,B 0,C 180,E1 11512.226,E2 11512.226} C_VEL
LIN {X 0,Y 365.999,Z 726.025,A -85,B 0,C 180,E1 11518.81,E2 11518.81} C_VEL
LIN {X 0,Y 365.596,Z 716.723,A -85,B 0,C 180,E1 11525.516,E2 11525.516} C_VEL
LIN {X 0,Y 367.1,Z 692.678,A -85,B 0,C 180,E1 11531.624,E2 11531.624} C_VEL
LIN {X 0,Y 369.803,Z 656.389,A -85,B 0,C 180,E1 11536.384,E2 11536.384} C_VEL
LIN {X 0,Y 368.202,Z 628.747,A -85,B 0,C 180,E1 11538.593,E2 11538.593} C_VEL
LIN {X 0,Y 362.248,Z 602.81,A -85,B 0,C 180,E1 11540.16,E2 11540.16} C_VEL
LIN {X 0,Y 361.49,Z 602.81,A -85,B 0,C 180,E1 11551.648,E2 11551.648} C_VEL
LIN {X 0,Y 361.315,Z 602.81,A -85,B 0,C 180,E1 11563.864,E2 11563.864} C_VEL
LIN {X 0,Y 361.332,Z 602.81,A -85,B 0,C 180,E1 11575.441,E2 11575.441} C_VEL
LIN {X 0,Y 361.595,Z 602.81,A -85,B 0,C 180,E1 11586.485,E2 11586.485} C_VEL
LIN {X 0,Y 362.192,Z 602.81,A -85,B 0,C 180,E1 11596.658,E2 11596.658} C_VEL
LIN {X 0,Y 363.404,Z 602.81,A -85,B 0,C 180,E1 11608.784,E2 11608.784} C_VEL
LIN {X 0,Y 362.537,Z 602.81,A -85,B 0,C 180,E1 11620.836,E2 11620.836} C_VEL
LIN {X 0,Y 362.045,Z 602.81,A -85,B 0,C 180,E1 11630.849,E2 11630.849} C_VEL
LIN {X 0,Y 361.631,Z 602.81,A -85,B 0,C 180,E1 11641.61,E2 11641.61} C_VEL
LIN {X 0,Y 361.397,Z 602.81,A -85,B 0,C 180,E1 11653.822,E2 11653.822} C_VEL
LIN {X 0,Y 361.383,Z 602.81,A -85,B 0,C 180,E1 11665.47,E2 11665.47} C_VEL
LIN {X 0,Y 361.735,Z 604.546,A -85,B 0,C 180,E1 11667.008,E2 11667.008} C_VEL
LIN {X 0,Y 379.713,Z 660.409,A -85,B 0,C 180,E1 11670.61,E2 11670.61} C_VEL
LIN {X 0,Y 373.863,Z 712.146,A -85,B 0,C 180,E1 11674.911,E2 11674.911} C_VEL
LIN {X 0,Y 368.337,Z 753.341,A -85,B 0,C 180,E1 11681.027,E2 11681.027} C_VEL
LIN {X 0,Y 364.759,Z 781.544,A -85,B 0,C 180,E1 11688.337,E2 11688.337} C_VEL
LIN {X 0,Y 363.675,Z 796.359,A -85,B 0,C 180,E1 11696.413,E2 11696.413} C_VEL
LIN {X 0,Y 363.797,Z 797.849,A -85,B 0,C 180,E1 11703.589,E2 11703.589} C_VEL
LIN {X 0,Y 365.531,Z 786.193,A -85,B 0,C 180,E1 11711.913,E2 11711.913} C_VEL
LIN {X 0,Y 370.384,Z 759.543,A -85,B 0,C 180,E1 11719.781,E2 11719.781} C_VEL
LIN {X 0,Y 378.122,Z 719.743,A -85,B 0,C 180,E1 11726.198,E2 11726.198} C_VEL
LIN {X 0,Y 386.348,Z 668.424,A -85,B 0,C 180,E1 11730.841,E2 11730.841} C_VEL
LIN {X 0,Y 381.684,Z 640.075,A -85,B 0,C 180,E1 11733.64,E2 11733.64} C_VEL
LIN {X 0,Y 369.316,Z 615.923,A -85,B 0,C 180,E1 11738.191,E2 11738.191} C_VEL
LIN {X 0,Y 363.873,Z 608.622,A -85,B 0,C 180,E1 11741.722,E2 11741.722} C_VEL
LIN {X 0,Y 364.373,Z 609.055,A -85,B 0,C 180,E1 11747.671,E2 11747.671} C_VEL
LIN {X 0,Y 371.618,Z 619.904,A -85,B 0,C 180,E1 11751.838,E2 11751.838} C_VEL
LIN {X 0,Y 384.634,Z 646.011,A -85,B 0,C 180,E1 11756.075,E2 11756.075} C_VEL
LIN {X 0,Y 387.702,Z 665.525,A -85,B 0,C 180,E1 11757.475,E2 11757.475} C_VEL
LIN {X 0,Y 379.575,Z 723.696,A -85,B 0,C 180,E1 11760.865,E2 11760.865} C_VEL
LIN {X 0,Y 371.418,Z 773.63,A -85,B 0,C 180,E1 11766.437,E2 11766.437} C_VEL
LIN {X 0,Y 365.932,Z 809.932,A -85,B 0,C 180,E1 11773.457,E2 11773.457} C_VEL
LIN {X 0,Y 363.801,Z 831.575,A -85,B 0,C 180,E1 11781.021,E2 11781.021} C_VEL
LIN {X 0,Y 363.899,Z 839.827,A -85,B 0,C 180,E1 11789.007,E2 11789.007} C_VEL
LIN {X 0,Y 363.72,Z 837.483,A -85,B 0,C 180,E1 11794.404,E2 11794.404} C_VEL
LIN {X 0,Y 356.087,Z 828.366,A -85,B 0,C 180,E1 11799.739,E2 11799.739} C_VEL
LIN {X 0,Y 358.386,Z 802.376,A -85,B 0,C 180,E1 11807.688,E2 11807.688} C_VEL
LIN {X 0,Y 363.589,Z 762.662,A -85,B 0,C 180,E1 11814.359,E2 11814.359} C_VEL
LIN {X 0,Y 372.567,Z 699.546,A -85,B 0,C 180,E1 11820.371,E2 11820.371} C_VEL
LIN {X 0,Y 375.844,Z 655.451,A -85,B 0,C 180,E1 11822.691,E2 11822.691} C_VEL
LIN {X 0,Y 364.251,Z 622.917,A -85,B 0,C 180,E1 11825.58,E2 11825.58} C_VEL
LIN {X 0,Y 353.44,Z 602.81,A -85,B 0,C 180,E1 11828.915,E2 11828.915} C_VEL
LIN {X 0,Y 353.36,Z 602.81,A -85,B 0,C 180,E1 11838.748,E2 11838.748} C_VEL
LIN {X 0,Y 353.5,Z 602.81,A -85,B 0,C 180,E1 11850.416,E2 11850.416} C_VEL
LIN {X 0,Y 353.986,Z 605.247,A -85,B 0,C 180,E1 11852.245,E2 11852.245} C_VEL
LIN {X 0,Y 368.402,Z 636.439,A -85,B 0,C 180,E1 11857.093,E2 11857.093} C_VEL
LIN {X 0,Y 370.434,Z 664.276,A -85,B 0,C 180,E1 11860.157,E2 11860.157} C_VEL
LIN {X 0,Y 364.697,Z 699.549,A -85,B 0,C 180,E1 11865.233,E2 11865.233} C_VEL
LIN {X 0,Y 360.075,Z 721.121,A -85,B 0,C 180,E1 11871.516,E2 11871.516} C_VEL
LIN {X 0,Y 358.138,Z 727.233,A -85,B 0,C 180,E1 11876.354,E2 11876.354} C_VEL
LIN {X 0,Y 357.575,Z 721.989,A -85,B 0,C 180,E1 11883.648,E2 11883.648} C_VEL
LIN {X 0,Y 358.785,Z 702.106,A -85,B 0,C 180,E1 11890.046,E2 11890.046} C_VEL
LIN {X 0,Y 361.319,Z 668.354,A -85,B 0,C 180,E1 11895.432,E2 11895.432} C_VEL
LIN {X 0,Y 361.251,Z 634.083,A -85,B 0,C 180,E1 11898.543,E2 11898.543} C_VEL
LIN {X 0,Y 354.19,Z 602.81,A -85,B 0,C 180,E1 11900.577,E2 11900.577} C_VEL
LIN {X 0,Y 353.349,Z 602.81,A -85,B 0,C 180,E1 11912.465,E2 11912.465} C_VEL
LIN {X 0,Y 353.251,Z 602.81,A -85,B 0,C 180,E1 11924.839,E2 11924.839} C_VEL
LIN {X 0,Y 353.308,Z 602.81,A -85,B 0,C 180,E1 11936.877,E2 11936.877} C_VEL
LIN {X 0,Y 353.626,Z 602.81,A -85,B 0,C 180,E1 11948.588,E2 11948.588} C_VEL
LIN {X 0,Y 354.402,Z 602.81,A -85,B 0,C 180,E1 11958.871,E2 11958.871} C_VEL
LIN {X 0,Y 355.412,Z 602.81,A -85,B 0,C 180,E1 11968.757,E2 11968.757} C_VEL
LIN {X 0,Y 354.698,Z 602.81,A -85,B 0,C 180,E1 11978.591,E2 11978.591} C_VEL
LIN {X 0,Y 354.089,Z 602.81,A -85,B 0,C 180,E1 11988.726,E2 11988.726} C_VEL
LIN {X 0,Y 353.63,Z 602.81,A -85,B 0,C 180,E1 11999.544,E2 11999.544} C_VEL
LIN {X 0,Y 353.421,Z 602.81,A -85,B 0,C 180,E1 12011.691,E2 12011.691} C_VEL
LIN {X 0,Y 353.352,Z 602.81,A -85,B 0,C 180,E1 12022.568,E2 12022.568} C_VEL
LIN {X 0,Y 353.736,Z 604.739,A -85,B 0,C 180,E1 12026.433,E2 12026.433} C_VEL
LIN {X 0,Y 371.968,Z 661.2,A -85,B 0,C 180,E1 12030.177,E2 12030.177} C_VEL
LIN {X 0,Y 366.106,Z 713.36,A -85,B 0,C 180,E1 12034.65,E2 12034.65} C_VEL
LIN {X 0,Y 360.364,Z 754.606,A -85,B 0,C 180,E1 12040.956,E2 12040.956} C_VEL
LIN {X 0,Y 356.825,Z 781.998,A -85,B 0,C 180,E1 12048.242,E2 12048.242} C_VEL
LIN {X 0,Y 355.684,Z 796.716,A -85,B 0,C 180,E1 12056.333,E2 12056.333} C_VEL
LIN {X 0,Y 355.835,Z 798.453,A -85,B 0,C 180,E1 12063.67,E2 12063.67} C_VEL
LIN {X 0,Y 357.809,Z 786.373,A -85,B 0,C 180,E1 12072.479,E2 12072.479} C_VEL
LIN {X 0,Y 363.158,Z 759.832,A -85,B 0,C 180,E1 12080.42,E2 12080.42} C_VEL
LIN {X 0,Y 371.657,Z 719.43,A -85,B 0,C 180,E1 12087.018,E2 12087.018} C_VEL
LIN {X 0,Y 380.549,Z 668.017,A -85,B 0,C 180,E1 12091.705,E2 12091.705} C_VEL
LIN {X 0,Y 374.608,Z 639.516,A -85,B 0,C 180,E1 12095.034,E2 12095.034} C_VEL
LIN {X 0,Y 363.773,Z 617.756,A -85,B 0,C 180,E1 12100.236,E2 12100.236} C_VEL
LIN {X 0,Y 361.018,Z 615.611,A -85,B 0,C 180,E1 12106.266,E2 12106.266} C_VEL
LIN {X 0,Y 365.537,Z 622.288,A -85,B 0,C 180,E1 12110.05,E2 12110.05} C_VEL
LIN {X 0,Y 376.175,Z 642.093,A -85,B 0,C 180,E1 12114.366,E2 12114.366} C_VEL
LIN {X 0,Y 382.055,Z 664.274,A -85,B 0,C 180,E1 12116.602,E2 12116.602} C_VEL
LIN {X 0,Y 372.996,Z 723.517,A -85,B 0,C 180,E1 12120.132,E2 12120.132} C_VEL
LIN {X 0,Y 364.123,Z 773.645,A -85,B 0,C 180,E1 12125.885,E2 12125.885} C_VEL
LIN {X 0,Y 358.215,Z 809.614,A -85,B 0,C 180,E1 12133.039,E2 12133.039} C_VEL
LIN {X 0,Y 355.771,Z 832.341,A -85,B 0,C 180,E1 12141.435,E2 12141.435} C_VEL
LIN {X 0,Y 355.956,Z 839.363,A -85,B 0,C 180,E1 12148.799,E2 12148.799} C_VEL
LIN {X 0,Y 355.66,Z 834.871,A -85,B 0,C 180,E1 12156.143,E2 12156.143} C_VEL
LIN {X 0,Y 356.087,Z 828.366,A -85,B 0,C 180,E1 12159.739,E2 12159.739} C_VEL
LIN {X 0,Y 349.003,Z 813.786,A -85,B 0,C 180,E1 12164.876,E2 12164.876} C_VEL
LIN {X 0,Y 353.208,Z 780.071,A -85,B 0,C 180,E1 12172.133,E2 12172.133} C_VEL
LIN {X 0,Y 362.332,Z 721.07,A -85,B 0,C 180,E1 12179.326,E2 12179.326} C_VEL
LIN {X 0,Y 370.07,Z 667.911,A -85,B 0,C 180,E1 12182.793,E2 12182.793} C_VEL
LIN {X 0,Y 362.911,Z 635.118,A -85,B 0,C 180,E1 12185.289,E2 12185.289} C_VEL
LIN {X 0,Y 347.555,Z 608.188,A -85,B 0,C 180,E1 12189.873,E2 12189.873} C_VEL
LIN {X 0,Y 345.413,Z 602.81,A -85,B 0,C 180,E1 12190.964,E2 12190.964} C_VEL
LIN {X 0,Y 345.303,Z 602.81,A -85,B 0,C 180,E1 12203.608,E2 12203.608} C_VEL
LIN {X 0,Y 345.688,Z 604.691,A -85,B 0,C 180,E1 12210.071,E2 12210.071} C_VEL
LIN {X 0,Y 360.009,Z 632.515,A -85,B 0,C 180,E1 12215.47,E2 12215.47} C_VEL
LIN {X 0,Y 364.385,Z 662.112,A -85,B 0,C 180,E1 12219.127,E2 12219.127} C_VEL
LIN {X 0,Y 358.203,Z 697.607,A -85,B 0,C 180,E1 12224.014,E2 12224.014} C_VEL
LIN {X 0,Y 352.859,Z 720.324,A -85,B 0,C 180,E1 12230.093,E2 12230.093} C_VEL
LIN {X 0,Y 350.291,Z 728.666,A -85,B 0,C 180,E1 12236.272,E2 12236.272} C_VEL
LIN {X 0,Y 349.66,Z 722.927,A -85,B 0,C 180,E1 12243.731,E2 12243.731} C_VEL
LIN {X 0,Y 350.896,Z 702.453,A -85,B 0,C 180,E1 12250.274,E2 12250.274} C_VEL
LIN {X 0,Y 353.57,Z 668.107,A -85,B 0,C 180,E1 12255.772,E2 12255.772} C_VEL
LIN {X 0,Y 353.234,Z 634.121,A -85,B 0,C 180,E1 12258.887,E2 12258.887} C_VEL
LIN {X 0,Y 346.168,Z 602.81,A -85,B 0,C 180,E1 12260.847,E2 12260.847} C_VEL
LIN {X 0,Y 345.294,Z 602.81,A -85,B 0,C 180,E1 12273.32,E2 12273.32} C_VEL
LIN {X 0,Y 345.136,Z 602.81,A -85,B 0,C 180,E1 12283.467,E2 12283.467} C_VEL
LIN {X 0,Y 345.254,Z 602.81,A -85,B 0,C 180,E1 12294.399,E2 12294.399} C_VEL
LIN {X 0,Y 345.494,Z 602.81,A -85,B 0,C 180,E1 12305.318,E2 12305.318} C_VEL
LIN {X 0,Y 346.126,Z 602.81,A -85,B 0,C 180,E1 12316.027,E2 12316.027} C_VEL
LIN {X 0,Y 347.392,Z 602.81,A -85,B 0,C 180,E1 12328.728,E2 12328.728} C_VEL
LIN {X 0,Y 346.511,Z 602.81,A -85,B 0,C 180,E1 12339.833,E2 12339.833} C_VEL
LIN {X 0,Y 345.951,Z 602.81,A -85,B 0,C 180,E1 12351.867,E2 12351.867} C_VEL
LIN {X 0,Y 345.443,Z 602.81,A -85,B 0,C 180,E1 12363.278,E2 12363.278} C_VEL
LIN {X 0,Y 345.242,Z 602.81,A -85,B 0,C 180,E1 12373.514,E2 12373.514} C_VEL
LIN {X 0,Y 345.465,Z 603.561,A -85,B 0,C 180,E1 12385.782,E2 12385.782} C_VEL
LIN {X 0,Y 363.892,Z 660.71,A -85,B 0,C 180,E1 12389.637,E2 12389.637} C_VEL
LIN {X 0,Y 358.784,Z 711.38,A -85,B 0,C 180,E1 12394.008,E2 12394.008} C_VEL
LIN {X 0,Y 352.957,Z 752.543,A -85,B 0,C 180,E1 12400.212,E2 12400.212} C_VEL
LIN {X 0,Y 348.959,Z 781.944,A -85,B 0,C 180,E1 12407.959,E2 12407.959} C_VEL
LIN {X 0,Y 347.691,Z 797.038,A -85,B 0,C 180,E1 12416.248,E2 12416.248} C_VEL
LIN {X 0,Y 347.858,Z 799.047,A -85,B 0,C 180,E1 12423.754,E2 12423.754} C_VEL
LIN {X 0,Y 349.788,Z 788.747,A -85,B 0,C 180,E1 12432.066,E2 12432.066} C_VEL
LIN {X 0,Y 355.343,Z 763.164,A -85,B 0,C 180,E1 12440.411,E2 12440.411} C_VEL
LIN {X 0,Y 364.376,Z 724.017,A -85,B 0,C 180,E1 12447.267,E2 12447.267} C_VEL
LIN {X 0,Y 374.091,Z 673.244,A -85,B 0,C 180,E1 12452.244,E2 12452.244} C_VEL
LIN {X 0,Y 371.287,Z 648.407,A -85,B 0,C 180,E1 12455.04,E2 12455.04} C_VEL
LIN {X 0,Y 362.092,Z 627.997,A -85,B 0,C 180,E1 12459.704,E2 12459.704} C_VEL
LIN {X 0,Y 358.403,Z 622.641,A -85,B 0,C 180,E1 12464.318,E2 12464.318} C_VEL
LIN {X 0,Y 361.913,Z 628.098,A -85,B 0,C 180,E1 12469.185,E2 12469.185} C_VEL
LIN {X 0,Y 371.348,Z 646.595,A -85,B 0,C 180,E1 12473.616,E2 12473.616} C_VEL
LIN {X 0,Y 376.32,Z 665.987,A -85,B 0,C 180,E1 12475.789,E2 12475.789} C_VEL
LIN {X 0,Y 366.243,Z 725.28,A -85,B 0,C 180,E1 12479.524,E2 12479.524} C_VEL
LIN {X 0,Y 356.596,Z 775.096,A -85,B 0,C 180,E1 12485.51,E2 12485.51} C_VEL
LIN {X 0,Y 350.398,Z 810.051,A -85,B 0,C 180,E1 12492.781,E2 12492.781} C_VEL
LIN {X 0,Y 347.791,Z 832.024,A -85,B 0,C 180,E1 12501.237,E2 12501.237} C_VEL
LIN {X 0,Y 347.958,Z 838.886,A -85,B 0,C 180,E1 12508.771,E2 12508.771} C_VEL
LIN {X 0,Y 347.663,Z 834.192,A -85,B 0,C 180,E1 12516.285,E2 12516.285} C_VEL
LIN {X 0,Y 348.716,Z 816.047,A -85,B 0,C 180,E1 12524.189,E2 12524.189} C_VEL
LIN {X 0,Y 349.003,Z 813.786,A -85,B 0,C 180,E1 12524.876,E2 12524.876} C_VEL
LIN {X 0,Y 343.224,Z 794.267,A -85,B 0,C 180,E1 12529.715,E2 12529.715} C_VEL
LIN {X 0,Y 350.503,Z 746.971,A -85,B 0,C 180,E1 12537.059,E2 12537.059} C_VEL
LIN {X 0,Y 359.762,Z 696.477,A -85,B 0,C 180,E1 12541.996,E2 12541.996} C_VEL
LIN {X 0,Y 363.055,Z 659.178,A -85,B 0,C 180,E1 12544.191,E2 12544.191} C_VEL
LIN {X 0,Y 353.88,Z 631.385,A -85,B 0,C 180,E1 12547.059,E2 12547.059} C_VEL
LIN {X 0,Y 340.186,Z 608.902,A -85,B 0,C 180,E1 12552.11,E2 12552.11} C_VEL
LIN {X 0,Y 337.168,Z 602.81,A -85,B 0,C 180,E1 12554.26,E2 12554.26} C_VEL
LIN {X 0,Y 337.414,Z 604.012,A -85,B 0,C 180,E1 12566.976,E2 12566.976} C_VEL
LIN {X 0,Y 348.89,Z 623.714,A -85,B 0,C 180,E1 12572.561,E2 12572.561} C_VEL
LIN {X 0,Y 357.943,Z 653.658,A -85,B 0,C 180,E1 12577.208,E2 12577.208} C_VEL
LIN {X 0,Y 352.253,Z 693.852,A -85,B 0,C 180,E1 12582.447,E2 12582.447} C_VEL
LIN {X 0,Y 346.132,Z 719.152,A -85,B 0,C 180,E1 12588.62,E2 12588.62} C_VEL
LIN {X 0,Y 343.104,Z 729.206,A -85,B 0,C 180,E1 12594.509,E2 12594.509} C_VEL
LIN {X 0,Y 341.454,Z 727.828,A -85,B 0,C 180,E1 12601.271,E2 12601.271} C_VEL
LIN {X 0,Y 342.028,Z 711.748,A -85,B 0,C 180,E1 12608.289,E2 12608.289} C_VEL
LIN {X 0,Y 344.62,Z 680.384,A -85,B 0,C 180,E1 12614.496,E2 12614.496} C_VEL
LIN {X 0,Y 346.346,Z 639.967,A -85,B 0,C 180,E1 12618.757,E2 12618.757} C_VEL
LIN {X 0,Y 338.08,Z 602.81,A -85,B 0,C 180,E1 12621.343,E2 12621.343} C_VEL
LIN {X 0,Y 337.223,Z 602.81,A -85,B 0,C 180,E1 12634.226,E2 12634.226} C_VEL
LIN {X 0,Y 337.058,Z 602.81,A -85,B 0,C 180,E1 12645.722,E2 12645.722} C_VEL
LIN {X 0,Y 337.256,Z 602.81,A -85,B 0,C 180,E1 12656.343,E2 12656.343} C_VEL
LIN {X 0,Y 337.515,Z 602.81,A -85,B 0,C 180,E1 12667.511,E2 12667.511} C_VEL
LIN {X 0,Y 338.288,Z 602.81,A -85,B 0,C 180,E1 12678.334,E2 12678.334} C_VEL
LIN {X 0,Y 339.379,Z 602.81,A -85,B 0,C 180,E1 12688.698,E2 12688.698} C_VEL
LIN {X 0,Y 338.624,Z 602.81,A -85,B 0,C 180,E1 12699.002,E2 12699.002} C_VEL
LIN {X 0,Y 337.99,Z 602.81,A -85,B 0,C 180,E1 12709.654,E2 12709.654} C_VEL
LIN {X 0,Y 337.444,Z 602.81,A -85,B 0,C 180,E1 12721.114,E2 12721.114} C_VEL
LIN {X 0,Y 337.185,Z 602.81,A -85,B 0,C 180,E1 12732.052,E2 12732.052} C_VEL
LIN {X 0,Y 337.329,Z 602.81,A -85,B 0,C 180,E1 12744.834,E2 12744.834} C_VEL
LIN {X 0,Y 356.877,Z 666.45,A -85,B 0,C 180,E1 12749.592,E2 12749.592} C_VEL
LIN {X 0,Y 350.318,Z 717.486,A -85,B 0,C 180,E1 12754.333,E2 12754.333} C_VEL
LIN {X 0,Y 344.326,Z 757.812,A -85,B 0,C 180,E1 12760.979,E2 12760.979} C_VEL
LIN {X 0,Y 340.579,Z 785.491,A -85,B 0,C 180,E1 12769.087,E2 12769.087} C_VEL
LIN {X 0,Y 339.646,Z 798.117,A -85,B 0,C 180,E1 12777.188,E2 12777.188} C_VEL
LIN {X 0,Y 339.904,Z 799.638,A -85,B 0,C 180,E1 12783.842,E2 12783.842} C_VEL
LIN {X 0,Y 341.974,Z 789.694,A -85,B 0,C 180,E1 12792.346,E2 12792.346} C_VEL
LIN {X 0,Y 348.057,Z 764.251,A -85,B 0,C 180,E1 12800.95,E2 12800.95} C_VEL
LIN {X 0,Y 357.836,Z 725.307,A -85,B 0,C 180,E1 12807.98,E2 12807.98} C_VEL
LIN {X 0,Y 368.512,Z 674.346,A -85,B 0,C 180,E1 12813.113,E2 12813.113} C_VEL
LIN {X 0,Y 365.836,Z 651.156,A -85,B 0,C 180,E1 12816.055,E2 12816.055} C_VEL
LIN {X 0,Y 358.394,Z 632.46,A -85,B 0,C 180,E1 12821.02,E2 12821.02} C_VEL
LIN {X 0,Y 357.328,Z 631.641,A -85,B 0,C 180,E1 12826.944,E2 12826.944} C_VEL
LIN {X 0,Y 364.419,Z 645.373,A -85,B 0,C 180,E1 12831.785,E2 12831.785} C_VEL
LIN {X 0,Y 370.863,Z 667.141,A -85,B 0,C 180,E1 12834.908,E2 12834.908} C_VEL
LIN {X 0,Y 359.595,Z 727.367,A -85,B 0,C 180,E1 12838.898,E2 12838.898} C_VEL
LIN {X 0,Y 349.313,Z 775.631,A -85,B 0,C 180,E1 12844.965,E2 12844.965} C_VEL
LIN {X 0,Y 342.456,Z 811.069,A -85,B 0,C 180,E1 12852.684,E2 12852.684} C_VEL
LIN {X 0,Y 339.82,Z 831.734,A -85,B 0,C 180,E1 12861.03,E2 12861.03} C_VEL
LIN {X 0,Y 339.974,Z 838.41,A -85,B 0,C 180,E1 12868.742,E2 12868.742} C_VEL
LIN {X 0,Y 339.696,Z 832.493,A -85,B 0,C 180,E1 12877.077,E2 12877.077} C_VEL
LIN {X 0,Y 341.104,Z 812.85,A -85,B 0,C 180,E1 12885.171,E2 12885.171} C_VEL
LIN {X 0,Y 343.224,Z 794.267,A -85,B 0,C 180,E1 12889.715,E2 12889.715} C_VEL
LIN {X 0,Y 339.042,Z 770.602,A -85,B 0,C 180,E1 12894.107,E2 12894.107} C_VEL
LIN {X 0,Y 349.086,Z 718.866,A -85,B 0,C 180,E1 12900.918,E2 12900.918} C_VEL
LIN {X 0,Y 357.184,Z 662.565,A -85,B 0,C 180,E1 12904.866,E2 12904.866} C_VEL
LIN {X 0,Y 348.921,Z 635.895,A -85,B 0,C 180,E1 12907.846,E2 12907.846} C_VEL
LIN {X 0,Y 336.69,Z 615.452,A -85,B 0,C 180,E1 12912.798,E2 12912.798} C_VEL
LIN {X 0,Y 331.52,Z 608.527,A -85,B 0,C 180,E1 12916.617,E2 12916.617} C_VEL
LIN {X 0,Y 331.079,Z 608.076,A -85,B 0,C 180,E1 12923.729,E2 12923.729} C_VEL
LIN {X 0,Y 335.378,Z 614.068,A -85,B 0,C 180,E1 12927.485,E2 12927.485} C_VEL
LIN {X 0,Y 346.06,Z 633.247,A -85,B 0,C 180,E1 12932.819,E2 12932.819} C_VEL
LIN {X 0,Y 351.978,Z 663.4,A -85,B 0,C 180,E1 12937.44,E2 12937.44} C_VEL
LIN {X 0,Y 344.41,Z 700.143,A -85,B 0,C 180,E1 12942.696,E2 12942.696} C_VEL
LIN {X 0,Y 338.062,Z 722.835,A -85,B 0,C 180,E1 12949,E2 12949} C_VEL
LIN {X 0,Y 334.627,Z 731.558,A -85,B 0,C 180,E1 12956.098,E2 12956.098} C_VEL
LIN {X 0,Y 333.751,Z 725.885,A -85,B 0,C 180,E1 12963.256,E2 12963.256} C_VEL
LIN {X 0,Y 334.879,Z 705.922,A -85,B 0,C 180,E1 12970.111,E2 12970.111} C_VEL
LIN {X 0,Y 337.693,Z 671.519,A -85,B 0,C 180,E1 12975.974,E2 12975.974} C_VEL
LIN {X 0,Y 337.737,Z 637.231,A -85,B 0,C 180,E1 12979.335,E2 12979.335} C_VEL
LIN {X 0,Y 330.044,Z 602.81,A -85,B 0,C 180,E1 12981.664,E2 12981.664} C_VEL
LIN {X 0,Y 329.259,Z 602.81,A -85,B 0,C 180,E1 12992.003,E2 12992.003} C_VEL
LIN {X 0,Y 329.053,Z 602.81,A -85,B 0,C 180,E1 13004.347,E2 13004.347} C_VEL
LIN {X 0,Y 329.062,Z 602.81,A -85,B 0,C 180,E1 13014.776,E2 13014.776} C_VEL
LIN {X 0,Y 329.478,Z 602.81,A -85,B 0,C 180,E1 13026.932,E2 13026.932} C_VEL
LIN {X 0,Y 330.242,Z 602.81,A -85,B 0,C 180,E1 13038.045,E2 13038.045} C_VEL
LIN {X 0,Y 331.358,Z 602.81,A -85,B 0,C 180,E1 13048.667,E2 13048.667} C_VEL
LIN {X 0,Y 330.581,Z 602.81,A -85,B 0,C 180,E1 13059.29,E2 13059.29} C_VEL
LIN {X 0,Y 329.928,Z 602.81,A -85,B 0,C 180,E1 13070.155,E2 13070.155} C_VEL
LIN {X 0,Y 329.359,Z 602.81,A -85,B 0,C 180,E1 13081.967,E2 13081.967} C_VEL
LIN {X 0,Y 329.166,Z 602.81,A -85,B 0,C 180,E1 13094.396,E2 13094.396} C_VEL
LIN {X 0,Y 329.508,Z 604.397,A -85,B 0,C 180,E1 13104.56,E2 13104.56} C_VEL
LIN {X 0,Y 348.448,Z 662.785,A -85,B 0,C 180,E1 13108.766,E2 13108.766} C_VEL
LIN {X 0,Y 343.297,Z 713.433,A -85,B 0,C 180,E1 13113.415,E2 13113.415} C_VEL
LIN {X 0,Y 337.082,Z 754.37,A -85,B 0,C 180,E1 13119.926,E2 13119.926} C_VEL
LIN {X 0,Y 332.836,Z 783.78,A -85,B 0,C 180,E1 13128.163,E2 13128.163} C_VEL
LIN {X 0,Y 331.729,Z 797.63,A -85,B 0,C 180,E1 13136.068,E2 13136.068} C_VEL
LIN {X 0,Y 331.928,Z 800.24,A -85,B 0,C 180,E1 13143.934,E2 13143.934} C_VEL
LIN {X 0,Y 334.184,Z 790.716,A -85,B 0,C 180,E1 13152.622,E2 13152.622} C_VEL
LIN {X 0,Y 340.686,Z 765.972,A -85,B 0,C 180,E1 13161.378,E2 13161.378} C_VEL
LIN {X 0,Y 351.42,Z 726.814,A -85,B 0,C 180,E1 13168.713,E2 13168.713} C_VEL
LIN {X 0,Y 363.08,Z 676.116,A -85,B 0,C 180,E1 13173.989,E2 13173.989} C_VEL
LIN {X 0,Y 360.736,Z 653.956,A -85,B 0,C 180,E1 13177.154,E2 13177.154} C_VEL
LIN {X 0,Y 355.305,Z 639.51,A -85,B 0,C 180,E1 13181.815,E2 13181.815} C_VEL
LIN {X 0,Y 355.903,Z 640.191,A -85,B 0,C 180,E1 13187.657,E2 13187.657} C_VEL
LIN {X 0,Y 363.092,Z 658.353,A -85,B 0,C 180,E1 13192.529,E2 13192.529} C_VEL
LIN {X 0,Y 364.891,Z 672.947,A -85,B 0,C 180,E1 13194.196,E2 13194.196} C_VEL
LIN {X 0,Y 352.676,Z 731.004,A -85,B 0,C 180,E1 13198.399,E2 13198.399} C_VEL
LIN {X 0,Y 341.649,Z 778.168,A -85,B 0,C 180,E1 13204.716,E2 13204.716} C_VEL
LIN {X 0,Y 334.303,Z 813.043,A -85,B 0,C 180,E1 13212.863,E2 13212.863} C_VEL
LIN {X 0,Y 331.856,Z 831.449,A -85,B 0,C 180,E1 13220.813,E2 13220.813} C_VEL
LIN {X 0,Y 331.977,Z 837.912,A -85,B 0,C 180,E1 13228.712,E2 13228.712} C_VEL
LIN {X 0,Y 331.718,Z 831.712,A -85,B 0,C 180,E1 13237.248,E2 13237.248} C_VEL
LIN {X 0,Y 333.263,Z 811.643,A -85,B 0,C 180,E1 13245.537,E2 13245.537} C_VEL
LIN {X 0,Y 338.151,Z 776.142,A -85,B 0,C 180,E1 13253.235,E2 13253.235} C_VEL
LIN {X 0,Y 339.042,Z 770.602,A -85,B 0,C 180,E1 13254.107,E2 13254.107} C_VEL
LIN {X 0,Y 336.419,Z 746.055,A -85,B 0,C 180,E1 13258.438,E2 13258.438} C_VEL
LIN {X 0,Y 347.23,Z 695.973,A -85,B 0,C 180,E1 13263.639,E2 13263.639} C_VEL
LIN {X 0,Y 350.978,Z 663.761,A -85,B 0,C 180,E1 13265.787,E2 13265.787} C_VEL
LIN {X 0,Y 343.682,Z 639.318,A -85,B 0,C 180,E1 13268.83,E2 13268.83} C_VEL
LIN {X 0,Y 332.414,Z 620.242,A -85,B 0,C 180,E1 13274.141,E2 13274.141} C_VEL
LIN {X 0,Y 327.757,Z 614.189,A -85,B 0,C 180,E1 13279.84,E2 13279.84} C_VEL
LIN {X 0,Y 331.966,Z 620.298,A -85,B 0,C 180,E1 13286.8,E2 13286.8} C_VEL
LIN {X 0,Y 341.669,Z 639.888,A -85,B 0,C 180,E1 13292.509,E2 13292.509} C_VEL
LIN {X 0,Y 345.528,Z 667.352,A -85,B 0,C 180,E1 13296.887,E2 13296.887} C_VEL
LIN {X 0,Y 337.275,Z 703.217,A -85,B 0,C 180,E1 13302.318,E2 13302.318} C_VEL
LIN {X 0,Y 330.497,Z 724.938,A -85,B 0,C 180,E1 13308.745,E2 13308.745} C_VEL
LIN {X 0,Y 326.793,Z 733.011,A -85,B 0,C 180,E1 13316.004,E2 13316.004} C_VEL
LIN {X 0,Y 325.835,Z 726.789,A -85,B 0,C 180,E1 13323.335,E2 13323.335} C_VEL
LIN {X 0,Y 327.027,Z 706.127,A -85,B 0,C 180,E1 13330.356,E2 13330.356} C_VEL
LIN {X 0,Y 329.932,Z 670.98,A -85,B 0,C 180,E1 13336.36,E2 13336.36} C_VEL
LIN {X 0,Y 329.86,Z 638.155,A -85,B 0,C 180,E1 13339.623,E2 13339.623} C_VEL
LIN {X 0,Y 321.976,Z 602.81,A -85,B 0,C 180,E1 13341.969,E2 13341.969} C_VEL
LIN {X 0,Y 321.043,Z 602.81,A -85,B 0,C 180,E1 13354.158,E2 13354.158} C_VEL
LIN {X 0,Y 320.986,Z 602.81,A -85,B 0,C 180,E1 13367.116,E2 13367.116} C_VEL
LIN {X 0,Y 321.07,Z 602.81,A -85,B 0,C 180,E1 13377.053,E2 13377.053} C_VEL
LIN {X 0,Y 321.507,Z 602.81,A -85,B 0,C 180,E1 13389.246,E2 13389.246} C_VEL
LIN {X 0,Y 322.462,Z 602.81,A -85,B 0,C 180,E1 13400.498,E2 13400.498} C_VEL
LIN {X 0,Y 323.015,Z 602.81,A -85,B 0,C 180,E1 13411.324,E2 13411.324} C_VEL
LIN {X 0,Y 322.304,Z 602.81,A -85,B 0,C 180,E1 13422.208,E2 13422.208} C_VEL
LIN {X 0,Y 321.695,Z 602.81,A -85,B 0,C 180,E1 13433.612,E2 13433.612} C_VEL
LIN {X 0,Y 321.217,Z 602.81,A -85,B 0,C 180,E1 13446.163,E2 13446.163} C_VEL
LIN {X 0,Y 321.071,Z 602.81,A -85,B 0,C 180,E1 13457.065,E2 13457.065} C_VEL
LIN {X 0,Y 321.509,Z 604.475,A -85,B 0,C 180,E1 13463.911,E2 13463.911} C_VEL
LIN {X 0,Y 340.378,Z 662.633,A -85,B 0,C 180,E1 13468.209,E2 13468.209} C_VEL
LIN {X 0,Y 337.201,Z 703.161,A -85,B 0,C 180,E1 13471.804,E2 13471.804} C_VEL
LIN {X 0,Y 330.644,Z 746.928,A -85,B 0,C 180,E1 13478.108,E2 13478.108} C_VEL
LIN {X 0,Y 325.946,Z 778.093,A -85,B 0,C 180,E1 13485.855,E2 13485.855} C_VEL
LIN {X 0,Y 323.829,Z 796.362,A -85,B 0,C 180,E1 13494.624,E2 13494.624} C_VEL
LIN {X 0,Y 323.457,Z 801.104,A -85,B 0,C 180,E1 13501.346,E2 13501.346} C_VEL
LIN {X 0,Y 325.66,Z 795.182,A -85,B 0,C 180,E1 13510.744,E2 13510.744} C_VEL
LIN {X 0,Y 331.728,Z 773.918,A -85,B 0,C 180,E1 13520.067,E2 13520.067} C_VEL
LIN {X 0,Y 342.08,Z 739.409,A -85,B 0,C 180,E1 13527.763,E2 13527.763} C_VEL
LIN {X 0,Y 354.837,Z 691.415,A -85,B 0,C 180,E1 13533.777,E2 13533.777} C_VEL
LIN {X 0,Y 358.137,Z 669.557,A -85,B 0,C 180,E1 13535.967,E2 13535.967} C_VEL
LIN {X 0,Y 354.482,Z 651.491,A -85,B 0,C 180,E1 13539.895,E2 13539.895} C_VEL
LIN {X 0,Y 351.973,Z 645.805,A -85,B 0,C 180,E1 13544.687,E2 13544.687} C_VEL
LIN {X 0,Y 355.047,Z 651.917,A -85,B 0,C 180,E1 13549.104,E2 13549.104} C_VEL
LIN {X 0,Y 360.312,Z 672.527,A -85,B 0,C 180,E1 13553.143,E2 13553.143} C_VEL
LIN {X 0,Y 346.827,Z 730.567,A -85,B 0,C 180,E1 13557.431,E2 13557.431} C_VEL
LIN {X 0,Y 334.473,Z 779.004,A -85,B 0,C 180,E1 13564.134,E2 13564.134} C_VEL
LIN {X 0,Y 326.591,Z 813.135,A -85,B 0,C 180,E1 13572.445,E2 13572.445} C_VEL
LIN {X 0,Y 323.928,Z 831.159,A -85,B 0,C 180,E1 13580.586,E2 13580.586} C_VEL
LIN {X 0,Y 324.001,Z 837.382,A -85,B 0,C 180,E1 13588.68,E2 13588.68} C_VEL
LIN {X 0,Y 323.773,Z 830.909,A -85,B 0,C 180,E1 13597.427,E2 13597.427} C_VEL
LIN {X 0,Y 325.676,Z 809.291,A -85,B 0,C 180,E1 13606.243,E2 13606.243} C_VEL
LIN {X 0,Y 330.752,Z 773.295,A -85,B 0,C 180,E1 13613.951,E2 13613.951} C_VEL
LIN {X 0,Y 336.419,Z 746.055,A -85,B 0,C 180,E1 13618.438,E2 13618.438} C_VEL
LIN {X 0,Y 335.837,Z 719.457,A -85,B 0,C 180,E1 13622.441,E2 13622.441} C_VEL
LIN {X 0,Y 345.354,Z 667.137,A -85,B 0,C 180,E1 13626.533,E2 13626.533} C_VEL
LIN {X 0,Y 339.095,Z 644.238,A -85,B 0,C 180,E1 13629.637,E2 13629.637} C_VEL
LIN {X 0,Y 329.035,Z 625.214,A -85,B 0,C 180,E1 13635.252,E2 13635.252} C_VEL
LIN {X 0,Y 325.936,Z 622.545,A -85,B 0,C 180,E1 13642.618,E2 13642.618} C_VEL
LIN {X 0,Y 331.165,Z 630.696,A -85,B 0,C 180,E1 13647.997,E2 13647.997} C_VEL
LIN {X 0,Y 339.044,Z 655.221,A -85,B 0,C 180,E1 13653.849,E2 13653.849} C_VEL
LIN {X 0,Y 337.418,Z 678.746,A -85,B 0,C 180,E1 13657.21,E2 13657.21} C_VEL
LIN {X 0,Y 328.598,Z 711.649,A -85,B 0,C 180,E1 13663.222,E2 13663.222} C_VEL
LIN {X 0,Y 321.688,Z 730.461,A -85,B 0,C 180,E1 13670.495,E2 13670.495} C_VEL
LIN {X 0,Y 318.637,Z 733.536,A -85,B 0,C 180,E1 13678.633,E2 13678.633} C_VEL
LIN {X 0,Y 318.037,Z 721.431,A -85,B 0,C 180,E1 13686.161,E2 13686.161} C_VEL
LIN {X 0,Y 319.875,Z 695.02,A -85,B 0,C 180,E1 13692.997,E2 13692.997} C_VEL
LIN {X 0,Y 323.272,Z 655.258,A -85,B 0,C 180,E1 13698.402,E2 13698.402} C_VEL
LIN {X 0,Y 316.046,Z 612.306,A -85,B 0,C 180,E1 13701.812,E2 13701.812} C_VEL
LIN {X 0,Y 313.911,Z 602.81,A -85,B 0,C 180,E1 13702.483,E2 13702.483} C_VEL
LIN {X 0,Y 313.072,Z 602.81,A -85,B 0,C 180,E1 13713.874,E2 13713.874} C_VEL
LIN {X 0,Y 312.847,Z 602.81,A -85,B 0,C 180,E1 13725.278,E2 13725.278} C_VEL
LIN {X 0,Y 313.044,Z 602.81,A -85,B 0,C 180,E1 13738.024,E2 13738.024} C_VEL
LIN {X 0,Y 313.547,Z 602.81,A -85,B 0,C 180,E1 13750.684,E2 13750.684} C_VEL
LIN {X 0,Y 314.557,Z 602.81,A -85,B 0,C 180,E1 13763.051,E2 13763.051} C_VEL
LIN {X 0,Y 315.006,Z 602.81,A -85,B 0,C 180,E1 13771.358,E2 13771.358} C_VEL
LIN {X 0,Y 314.246,Z 602.81,A -85,B 0,C 180,E1 13782.527,E2 13782.527} C_VEL
LIN {X 0,Y 313.582,Z 602.81,A -85,B 0,C 180,E1 13794.262,E2 13794.262} C_VEL
LIN {X 0,Y 313.13,Z 602.81,A -85,B 0,C 180,E1 13807.252,E2 13807.252} C_VEL
LIN {X 0,Y 312.961,Z 602.81,A -85,B 0,C 180,E1 13819.115,E2 13819.115} C_VEL
LIN {X 0,Y 313.416,Z 604.575,A -85,B 0,C 180,E1 13823.241,E2 13823.241} C_VEL
LIN {X 0,Y 332.617,Z 663.48,A -85,B 0,C 180,E1 13827.738,E2 13827.738} C_VEL
LIN {X 0,Y 331.206,Z 693.427,A -85,B 0,C 180,E1 13830.355,E2 13830.355} C_VEL
LIN {X 0,Y 323.978,Z 740.291,A -85,B 0,C 180,E1 13836.541,E2 13836.541} C_VEL
LIN {X 0,Y 318.553,Z 774.593,A -85,B 0,C 180,E1 13844.46,E2 13844.46} C_VEL
LIN {X 0,Y 316.048,Z 794.617,A -85,B 0,C 180,E1 13853.108,E2 13853.108} C_VEL
LIN {X 0,Y 315.474,Z 801.584,A -85,B 0,C 180,E1 13861.38,E2 13861.38} C_VEL
LIN {X 0,Y 317.841,Z 796.109,A -85,B 0,C 180,E1 13871.012,E2 13871.012} C_VEL
LIN {X 0,Y 324.355,Z 775.449,A -85,B 0,C 180,E1 13880.544,E2 13880.544} C_VEL
LIN {X 0,Y 335.381,Z 742.013,A -85,B 0,C 180,E1 13888.367,E2 13888.367} C_VEL
LIN {X 0,Y 349.279,Z 694.755,A -85,B 0,C 180,E1 13894.579,E2 13894.579} C_VEL
LIN {X 0,Y 353.326,Z 673.362,A -85,B 0,C 180,E1 13896.823,E2 13896.823} C_VEL
LIN {X 0,Y 350.541,Z 656.147,A -85,B 0,C 180,E1 13901.276,E2 13901.276} C_VEL
LIN {X 0,Y 350.488,Z 654.669,A -85,B 0,C 180,E1 13906.837,E2 13906.837} C_VEL
LIN {X 0,Y 354.9,Z 670.736,A -85,B 0,C 180,E1 13911.509,E2 13911.509} C_VEL
LIN {X 0,Y 353.361,Z 684.04,A -85,B 0,C 180,E1 13912.69,E2 13912.69} C_VEL
LIN {X 0,Y 338.592,Z 739.942,A -85,B 0,C 180,E1 13917.493,E2 13917.493} C_VEL
LIN {X 0,Y 325.498,Z 786.253,A -85,B 0,C 180,E1 13924.798,E2 13924.798} C_VEL
LIN {X 0,Y 317.955,Z 817.098,A -85,B 0,C 180,E1 13933.396,E2 13933.396} C_VEL
LIN {X 0,Y 315.851,Z 832.69,A -85,B 0,C 180,E1 13941.736,E2 13941.736} C_VEL
LIN {X 0,Y 316.007,Z 836.843,A -85,B 0,C 180,E1 13948.647,E2 13948.647} C_VEL
LIN {X 0,Y 315.804,Z 830.079,A -85,B 0,C 180,E1 13957.615,E2 13957.615} C_VEL
LIN {X 0,Y 317.82,Z 808.327,A -85,B 0,C 180,E1 13966.551,E2 13966.551} C_VEL
LIN {X 0,Y 325.773,Z 761.369,A -85,B 0,C 180,E1 13976.623,E2 13976.623} C_VEL
LIN {X 0,Y 335.837,Z 719.457,A -85,B 0,C 180,E1 13982.441,E2 13982.441} C_VEL
LIN {X 0,Y 336.642,Z 690.373,A -85,B 0,C 180,E1 13985.89,E2 13985.89} C_VEL
LIN {X 0,Y 339.448,Z 667.348,A -85,B 0,C 180,E1 13987.661,E2 13987.661} C_VEL
LIN {X 0,Y 333.03,Z 645.792,A -85,B 0,C 180,E1 13991.247,E2 13991.247} C_VEL
LIN {X 0,Y 325.156,Z 631.731,A -85,B 0,C 180,E1 13996.717,E2 13996.717} C_VEL
LIN {X 0,Y 324.172,Z 631.107,A -85,B 0,C 180,E1 14003.689,E2 14003.689} C_VEL
LIN {X 0,Y 330.307,Z 644.914,A -85,B 0,C 180,E1 14009.885,E2 14009.885} C_VEL
LIN {X 0,Y 333.863,Z 669.995,A -85,B 0,C 180,E1 14014.956,E2 14014.956} C_VEL
LIN {X 0,Y 323.951,Z 706.602,A -85,B 0,C 180,E1 14020.856,E2 14020.856} C_VEL
LIN {X 0,Y 315.405,Z 729.173,A -85,B 0,C 180,E1 14028.199,E2 14028.199} C_VEL
LIN {X 0,Y 311.119,Z 735.845,A -85,B 0,C 180,E1 14035.802,E2 14035.802} C_VEL
LIN {X 0,Y 309.97,Z 728.409,A -85,B 0,C 180,E1 14043.506,E2 14043.506} C_VEL
LIN {X 0,Y 311.294,Z 706.398,A -85,B 0,C 180,E1 14050.886,E2 14050.886} C_VEL
LIN {X 0,Y 314.349,Z 670.687,A -85,B 0,C 180,E1 14057.015,E2 14057.015} C_VEL
LIN {X 0,Y 314.072,Z 639.722,A -85,B 0,C 180,E1 14060.2,E2 14060.2} C_VEL
LIN {X 0,Y 305.854,Z 602.81,A -85,B 0,C 180,E1 14062.805,E2 14062.805} C_VEL
LIN {X 0,Y 304.947,Z 602.81,A -85,B 0,C 180,E1 14074.905,E2 14074.905} C_VEL
LIN {X 0,Y 304.762,Z 602.81,A -85,B 0,C 180,E1 14087.736,E2 14087.736} C_VEL
LIN {X 0,Y 305.057,Z 602.81,A -85,B 0,C 180,E1 14100.515,E2 14100.515} C_VEL
LIN {X 0,Y 305.595,Z 602.81,A -85,B 0,C 180,E1 14111.147,E2 14111.147} C_VEL
LIN {X 0,Y 306.541,Z 602.81,A -85,B 0,C 180,E1 14122.868,E2 14122.868} C_VEL
LIN {X 0,Y 306.995,Z 602.81,A -85,B 0,C 180,E1 14131.393,E2 14131.393} C_VEL
LIN {X 0,Y 306.188,Z 602.81,A -85,B 0,C 180,E1 14142.862,E2 14142.862} C_VEL
LIN {X 0,Y 305.533,Z 602.81,A -85,B 0,C 180,E1 14154.944,E2 14154.944} C_VEL
LIN {X 0,Y 305.089,Z 602.81,A -85,B 0,C 180,E1 14164.858,E2 14164.858} C_VEL
LIN {X 0,Y 304.853,Z 602.81,A -85,B 0,C 180,E1 14177.782,E2 14177.782} C_VEL
LIN {X 0,Y 305.199,Z 603.942,A -85,B 0,C 180,E1 14182.508,E2 14182.508} C_VEL
LIN {X 0,Y 324.699,Z 663.796,A -85,B 0,C 180,E1 14187.203,E2 14187.203} C_VEL
LIN {X 0,Y 324.869,Z 685.067,A -85,B 0,C 180,E1 14189.086,E2 14189.086} C_VEL
LIN {X 0,Y 317.239,Z 734.304,A -85,B 0,C 180,E1 14195.137,E2 14195.137} C_VEL
LIN {X 0,Y 311.105,Z 770.598,A -85,B 0,C 180,E1 14202.985,E2 14202.985} C_VEL
LIN {X 0,Y 308.273,Z 793.62,A -85,B 0,C 180,E1 14212.222,E2 14212.222} C_VEL
LIN {X 0,Y 307.508,Z 802.061,A -85,B 0,C 180,E1 14221.416,E2 14221.416} C_VEL
LIN {X 0,Y 309.914,Z 797.377,A -85,B 0,C 180,E1 14231.051,E2 14231.051} C_VEL
LIN {X 0,Y 316.642,Z 778.254,A -85,B 0,C 180,E1 14240.635,E2 14240.635} C_VEL
LIN {X 0,Y 328.764,Z 744.733,A -85,B 0,C 180,E1 14248.992,E2 14248.992} C_VEL
LIN {X 0,Y 344.022,Z 697.99,A -85,B 0,C 180,E1 14255.445,E2 14255.445} C_VEL
LIN {X 0,Y 348.769,Z 677.631,A -85,B 0,C 180,E1 14257.654,E2 14257.654} C_VEL
LIN {X 0,Y 347.453,Z 662.522,A -85,B 0,C 180,E1 14261.925,E2 14261.925} C_VEL
LIN {X 0,Y 347.767,Z 662.716,A -85,B 0,C 180,E1 14266.892,E2 14266.892} C_VEL
LIN {X 0,Y 350.825,Z 677.992,A -85,B 0,C 180,E1 14271.186,E2 14271.186} C_VEL
LIN {X 0,Y 334.103,Z 736.194,A -85,B 0,C 180,E1 14276.026,E2 14276.026} C_VEL
LIN {X 0,Y 319.713,Z 782.598,A -85,B 0,C 180,E1 14283.225,E2 14283.225} C_VEL
LIN {X 0,Y 310.717,Z 815.327,A -85,B 0,C 180,E1 14292.247,E2 14292.247} C_VEL
LIN {X 0,Y 307.879,Z 832.381,A -85,B 0,C 180,E1 14301.521,E2 14301.521} C_VEL
LIN {X 0,Y 308.021,Z 836.305,A -85,B 0,C 180,E1 14308.612,E2 14308.612} C_VEL
LIN {X 0,Y 307.855,Z 829.215,A -85,B 0,C 180,E1 14317.813,E2 14317.813} C_VEL
LIN {X 0,Y 310.011,Z 807.115,A -85,B 0,C 180,E1 14326.934,E2 14326.934} C_VEL
LIN {X 0,Y 321.715,Z 749.033,A -85,B 0,C 180,E1 14339.422,E2 14339.422} C_VEL
LIN {X 0,Y 334.208,Z 700.701,A -85,B 0,C 180,E1 14345.086,E2 14345.086} C_VEL
LIN {X 0,Y 336.642,Z 690.373,A -85,B 0,C 180,E1 14345.89,E2 14345.89} C_VEL
LIN {X 0,Y 334.186,Z 671.54,A -85,B 0,C 180,E1 14348.396,E2 14348.396} C_VEL
LIN {X 0,Y 328.807,Z 650.864,A -85,B 0,C 180,E1 14352.11,E2 14352.11} C_VEL
LIN {X 0,Y 322.295,Z 638.731,A -85,B 0,C 180,E1 14357.523,E2 14357.523} C_VEL
LIN {X 0,Y 322.337,Z 639.488,A -85,B 0,C 180,E1 14364.647,E2 14364.647} C_VEL
LIN {X 0,Y 327.628,Z 658.087,A -85,B 0,C 180,E1 14371.225,E2 14371.225} C_VEL
LIN {X 0,Y 326.667,Z 679.545,A -85,B 0,C 180,E1 14375.018,E2 14375.018} C_VEL
LIN {X 0,Y 316.046,Z 712.623,A -85,B 0,C 180,E1 14381.087,E2 14381.087} C_VEL
LIN {X 0,Y 307.322,Z 732.459,A -85,B 0,C 180,E1 14388.606,E2 14388.606} C_VEL
LIN {X 0,Y 303.286,Z 737.253,A -85,B 0,C 180,E1 14395.694,E2 14395.694} C_VEL
LIN {X 0,Y 302.019,Z 729.132,A -85,B 0,C 180,E1 14403.599,E2 14403.599} C_VEL
LIN {X 0,Y 303.396,Z 706.429,A -85,B 0,C 180,E1 14411.173,E2 14411.173} C_VEL
LIN {X 0,Y 306.629,Z 669.703,A -85,B 0,C 180,E1 14417.457,E2 14417.457} C_VEL
LIN {X 0,Y 306.256,Z 641.062,A -85,B 0,C 180,E1 14420.449,E2 14420.449} C_VEL
LIN {X 0,Y 297.691,Z 602.81,A -85,B 0,C 180,E1 14423.463,E2 14423.463} C_VEL
LIN {X 0,Y 296.777,Z 602.81,A -85,B 0,C 180,E1 14436.013,E2 14436.013} C_VEL
LIN {X 0,Y 296.747,Z 602.81,A -85,B 0,C 180,E1 14447.855,E2 14447.855} C_VEL
LIN {X 0,Y 297.073,Z 602.81,A -85,B 0,C 180,E1 14460.945,E2 14460.945} C_VEL
LIN {X 0,Y 297.724,Z 602.81,A -85,B 0,C 180,E1 14473.697,E2 14473.697} C_VEL
LIN {X 0,Y 298.77,Z 602.81,A -85,B 0,C 180,E1 14485.607,E2 14485.607} C_VEL
LIN {X 0,Y 298.617,Z 602.81,A -85,B 0,C 180,E1 14497.741,E2 14497.741} C_VEL
LIN {X 0,Y 297.758,Z 602.81,A -85,B 0,C 180,E1 14509.476,E2 14509.476} C_VEL
LIN {X 0,Y 297.037,Z 602.81,A -85,B 0,C 180,E1 14522.553,E2 14522.553} C_VEL
LIN {X 0,Y 296.87,Z 602.81,A -85,B 0,C 180,E1 14533.598,E2 14533.598} C_VEL
LIN {X 0,Y 297.045,Z 603.555,A -85,B 0,C 180,E1 14541.762,E2 14541.762} C_VEL
LIN {X 0,Y 316.814,Z 664.312,A -85,B 0,C 180,E1 14546.673,E2 14546.673} C_VEL
LIN {X 0,Y 317.405,Z 684.771,A -85,B 0,C 180,E1 14548.554,E2 14548.554} C_VEL
LIN {X 0,Y 309.686,Z 733.539,A -85,B 0,C 180,E1 14554.615,E2 14554.615} C_VEL
LIN {X 0,Y 303.262,Z 770.297,A -85,B 0,C 180,E1 14562.628,E2 14562.628} C_VEL
LIN {X 0,Y 300.323,Z 793.615,A -85,B 0,C 180,E1 14572.015,E2 14572.015} C_VEL
LIN {X 0,Y 299.525,Z 802.536,A -85,B 0,C 180,E1 14581.454,E2 14581.454} C_VEL
LIN {X 0,Y 301.526,Z 799.585,A -85,B 0,C 180,E1 14590.147,E2 14590.147} C_VEL
LIN {X 0,Y 308.172,Z 783.042,A -85,B 0,C 180,E1 14599.944,E2 14599.944} C_VEL
LIN {X 0,Y 320.415,Z 752.166,A -85,B 0,C 180,E1 14608.724,E2 14608.724} C_VEL
LIN {X 0,Y 336.876,Z 707.685,A -85,B 0,C 180,E1 14615.649,E2 14615.649} C_VEL
LIN {X 0,Y 344.481,Z 680.929,A -85,B 0,C 180,E1 14618.722,E2 14618.722} C_VEL
LIN {X 0,Y 344.213,Z 669.463,A -85,B 0,C 180,E1 14622.492,E2 14622.492} C_VEL
LIN {X 0,Y 345.001,Z 671.602,A -85,B 0,C 180,E1 14627.385,E2 14627.385} C_VEL
LIN {X 0,Y 345.97,Z 683.008,A -85,B 0,C 180,E1 14630.28,E2 14630.28} C_VEL
LIN {X 0,Y 327.894,Z 739.313,A -85,B 0,C 180,E1 14635.292,E2 14635.292} C_VEL
LIN {X 0,Y 312.148,Z 785.274,A -85,B 0,C 180,E1 14642.914,E2 14642.914} C_VEL
LIN {X 0,Y 302.773,Z 816.37,A -85,B 0,C 180,E1 14652.125,E2 14652.125} C_VEL
LIN {X 0,Y 299.878,Z 832.484,A -85,B 0,C 180,E1 14661.669,E2 14661.669} C_VEL
LIN {X 0,Y 300.026,Z 835.759,A -85,B 0,C 180,E1 14668.575,E2 14668.575} C_VEL
LIN {X 0,Y 299.837,Z 829.344,A -85,B 0,C 180,E1 14677.292,E2 14677.292} C_VEL
LIN {X 0,Y 301.749,Z 808.487,A -85,B 0,C 180,E1 14686.503,E2 14686.503} C_VEL
LIN {X 0,Y 313.995,Z 751.941,A -85,B 0,C 180,E1 14699.717,E2 14699.717} C_VEL
LIN {X 0,Y 327.604,Z 704.237,A -85,B 0,C 180,E1 14705.771,E2 14705.771} C_VEL
LIN {X 0,Y 334.186,Z 671.54,A -85,B 0,C 180,E1 14708.396,E2 14708.396} C_VEL
LIN {X 0,Y 329.619,Z 661.255,A -85,B 0,C 180,E1 14710.721,E2 14710.721} C_VEL
LIN {X 0,Y 323.847,Z 654.153,A -85,B 0,C 180,E1 14713.571,E2 14713.571} C_VEL
LIN {X 0,Y 319.999,Z 646.575,A -85,B 0,C 180,E1 14717.338,E2 14717.338} C_VEL
LIN {X 0,Y 318.839,Z 646.133,A -85,B 0,C 180,E1 14723.49,E2 14723.49} C_VEL
LIN {X 0,Y 322.178,Z 659.069,A -85,B 0,C 180,E1 14729.448,E2 14729.448} C_VEL
LIN {X 0,Y 321.694,Z 680.17,A -85,B 0,C 180,E1 14733.855,E2 14733.855} C_VEL
LIN {X 0,Y 309.521,Z 714.577,A -85,B 0,C 180,E1 14740.3,E2 14740.3} C_VEL
LIN {X 0,Y 300.376,Z 733.525,A -85,B 0,C 180,E1 14747.599,E2 14747.599} C_VEL
LIN {X 0,Y 295.461,Z 738.661,A -85,B 0,C 180,E1 14755.579,E2 14755.579} C_VEL
LIN {X 0,Y 294.088,Z 729.84,A -85,B 0,C 180,E1 14763.696,E2 14763.696} C_VEL
LIN {X 0,Y 295.507,Z 706.673,A -85,B 0,C 180,E1 14771.406,E2 14771.406} C_VEL
LIN {X 0,Y 298.788,Z 669.977,A -85,B 0,C 180,E1 14777.739,E2 14777.739} C_VEL
LIN {X 0,Y 298.1,Z 640.703,A -85,B 0,C 180,E1 14780.848,E2 14780.848} C_VEL
LIN {X 0,Y 289.665,Z 602.81,A -85,B 0,C 180,E1 14783.749,E2 14783.749} C_VEL
LIN {X 0,Y 288.745,Z 602.81,A -85,B 0,C 180,E1 14797.181,E2 14797.181} C_VEL
LIN {X 0,Y 288.73,Z 602.81,A -85,B 0,C 180,E1 14809.644,E2 14809.644} C_VEL
LIN {X 0,Y 289.084,Z 602.81,A -85,B 0,C 180,E1 14823.475,E2 14823.475} C_VEL
LIN {X 0,Y 289.91,Z 602.81,A -85,B 0,C 180,E1 14836.352,E2 14836.352} C_VEL
LIN {X 0,Y 291.277,Z 602.81,A -85,B 0,C 180,E1 14848.483,E2 14848.483} C_VEL
LIN {X 0,Y 290.36,Z 602.81,A -85,B 0,C 180,E1 14860.514,E2 14860.514} C_VEL
LIN {X 0,Y 289.461,Z 602.81,A -85,B 0,C 180,E1 14873.454,E2 14873.454} C_VEL
LIN {X 0,Y 288.88,Z 602.81,A -85,B 0,C 180,E1 14887.129,E2 14887.129} C_VEL
LIN {X 0,Y 288.935,Z 602.81,A -85,B 0,C 180,E1 14900.949,E2 14900.949} C_VEL
LIN {X 0,Y 308.812,Z 664.317,A -85,B 0,C 180,E1 14906.08,E2 14906.08} C_VEL
LIN {X 0,Y 310.172,Z 682.925,A -85,B 0,C 180,E1 14907.868,E2 14907.868} C_VEL
LIN {X 0,Y 302.049,Z 733.03,A -85,B 0,C 180,E1 14914.125,E2 14914.125} C_VEL
LIN {X 0,Y 295.297,Z 770.99,A -85,B 0,C 180,E1 14922.558,E2 14922.558} C_VEL
LIN {X 0,Y 292.349,Z 793.692,A -85,B 0,C 180,E1 14931.873,E2 14931.873} C_VEL
LIN {X 0,Y 291.542,Z 803.008,A -85,B 0,C 180,E1 14941.494,E2 14941.494} C_VEL
LIN {X 0,Y 294.57,Z 798.66,A -85,B 0,C 180,E1 14952.297,E2 14952.297} C_VEL
LIN {X 0,Y 303.271,Z 778.658,A -85,B 0,C 180,E1 14962.819,E2 14962.819} C_VEL
LIN {X 0,Y 318.603,Z 744.078,A -85,B 0,C 180,E1 14971.598,E2 14971.598} C_VEL
LIN {X 0,Y 337.168,Z 696.872,A -85,B 0,C 180,E1 14978.136,E2 14978.136} C_VEL
LIN {X 0,Y 340.596,Z 683.802,A -85,B 0,C 180,E1 14980.02,E2 14980.02} C_VEL
LIN {X 0,Y 340.811,Z 676.396,A -85,B 0,C 180,E1 14983.644,E2 14983.644} C_VEL
LIN {X 0,Y 341.906,Z 680.453,A -85,B 0,C 180,E1 14987.805,E2 14987.805} C_VEL
LIN {X 0,Y 341.225,Z 688.358,A -85,B 0,C 180,E1 14989.35,E2 14989.35} C_VEL
LIN {X 0,Y 320.842,Z 744.816,A -85,B 0,C 180,E1 14994.83,E2 14994.83} C_VEL
LIN {X 0,Y 304.055,Z 789.409,A -85,B 0,C 180,E1 15002.937,E2 15002.937} C_VEL
LIN {X 0,Y 294.345,Z 819.017,A -85,B 0,C 180,E1 15012.716,E2 15012.716} C_VEL
LIN {X 0,Y 291.836,Z 833.117,A -85,B 0,C 180,E1 15022.556,E2 15022.556} C_VEL
LIN {X 0,Y 291.941,Z 834.276,A -85,B 0,C 180,E1 15031.513,E2 15031.513} C_VEL
LIN {X 0,Y 292.273,Z 821.829,A -85,B 0,C 180,E1 15041.251,E2 15041.251} C_VEL
LIN {X 0,Y 295.415,Z 795.114,A -85,B 0,C 180,E1 15050.311,E2 15050.311} C_VEL
LIN {X 0,Y 308.313,Z 748.537,A -85,B 0,C 180,E1 15061.142,E2 15061.142} C_VEL
LIN {X 0,Y 323.148,Z 700.346,A -85,B 0,C 180,E1 15067.158,E2 15067.158} C_VEL
LIN {X 0,Y 328.792,Z 671.95,A -85,B 0,C 180,E1 15069.64,E2 15069.64} C_VEL
LIN {X 0,Y 323.847,Z 654.153,A -85,B 0,C 180,E1 15073.571,E2 15073.571} C_VEL
LIN {X 0,Y 319.337,Z 651.23,A -85,B 0,C 180,E1 15076.571,E2 15076.571} C_VEL
LIN {X 0,Y 315.944,Z 652.697,A -85,B 0,C 180,E1 15079.836,E2 15079.836} C_VEL
LIN {X 0,Y 316.433,Z 656.888,A -85,B 0,C 180,E1 15085.684,E2 15085.684} C_VEL
LIN {X 0,Y 317.873,Z 675.219,A -85,B 0,C 180,E1 15091.517,E2 15091.517} C_VEL
LIN {X 0,Y 304.221,Z 714.208,A -85,B 0,C 180,E1 15098.797,E2 15098.797} C_VEL
LIN {X 0,Y 293.581,Z 734.643,A -85,B 0,C 180,E1 15106.548,E2 15106.548} C_VEL
LIN {X 0,Y 287.63,Z 740.017,A -85,B 0,C 180,E1 15115.459,E2 15115.459} C_VEL
LIN {X 0,Y 286.142,Z 730.505,A -85,B 0,C 180,E1 15123.799,E2 15123.799} C_VEL
LIN {X 0,Y 287.666,Z 705.344,A -85,B 0,C 180,E1 15131.98,E2 15131.98} C_VEL
LIN {X 0,Y 291.19,Z 667.178,A -85,B 0,C 180,E1 15138.415,E2 15138.415} C_VEL
LIN {X 0,Y 289.759,Z 639.557,A -85,B 0,C 180,E1 15141.338,E2 15141.338} C_VEL
LIN {X 0,Y 281.597,Z 602.81,A -85,B 0,C 180,E1 15144.246,E2 15144.246} C_VEL
LIN {X 0,Y 280.647,Z 602.81,A -85,B 0,C 180,E1 15158.445,E2 15158.445} C_VEL
LIN {X 0,Y 280.64,Z 602.81,A -85,B 0,C 180,E1 15171.628,E2 15171.628} C_VEL
LIN {X 0,Y 281.003,Z 602.81,A -85,B 0,C 180,E1 15182.998,E2 15182.998} C_VEL
LIN {X 0,Y 281.857,Z 602.81,A -85,B 0,C 180,E1 15195.954,E2 15195.954} C_VEL
LIN {X 0,Y 283.25,Z 602.81,A -85,B 0,C 180,E1 15208.44,E2 15208.44} C_VEL
LIN {X 0,Y 282.308,Z 602.81,A -85,B 0,C 180,E1 15220.817,E2 15220.817} C_VEL
LIN {X 0,Y 281.405,Z 602.81,A -85,B 0,C 180,E1 15233.826,E2 15233.826} C_VEL
LIN {X 0,Y 280.874,Z 602.81,A -85,B 0,C 180,E1 15244.527,E2 15244.527} C_VEL
LIN {X 0,Y 280.662,Z 602.81,A -85,B 0,C 180,E1 15257.483,E2 15257.483} C_VEL
LIN {X 0,Y 281.164,Z 604.933,A -85,B 0,C 180,E1 15260.326,E2 15260.326} C_VEL
LIN {X 0,Y 300.562,Z 663.55,A -85,B 0,C 180,E1 15265.396,E2 15265.396} C_VEL
LIN {X 0,Y 302.523,Z 684.102,A -85,B 0,C 180,E1 15267.452,E2 15267.452} C_VEL
LIN {X 0,Y 294.259,Z 733.535,A -85,B 0,C 180,E1 15273.799,E2 15273.799} C_VEL
